// TwinCAT 3 PLC project P1_CompPP
// ProgramVersion: 3.1.4023.0
// libraries:
//   Tc2_Standard, * (Beckhoff Automation GmbH)
//   Tc2_System, * (Beckhoff Automation GmbH)
//   Tc2_Utilities, * (Beckhoff Automation GmbH)
//   Tc3_EventLogger, * (Beckhoff Automation GmbH)
//   Tc3_Module, * (Beckhoff Automation GmbH)
//   Tc2_Utilities,3.3.52.0,Beckhoff Automation GmbH
// project tree:
//   DUTs/ E_ChargerType.TcDUT (not stored), E_State.TcDUT, ST_Alarm_Base.TcDUT (not stored), ST_Charger_Base.TcDUT, ST_ChargeTime.TcDUT (not stored), ST_CSV_Record.TcDUT (not stored), ST_Module.TcDUT, ST_PB_Base.TcDUT (not stored), ST_PrefireDiscon_Base.TcDUT, ST_Segment_Base.TcDUT, ST_Setpoints_Base.TcDUT
//   GVLs/ Alarms_DB.TcGVL (not stored), ChargeTime_DB.TcGVL, csv_DB.TcGVL, EngVal.TcGVL, GVL.TcGVL, HMI_DB.TcGVL, Input.TcGVL, LCP1_IO.TcGVL, LCP2_IO.TcGVL, MCP_IO.TcGVL, Output.TcGVL, Permissives_DB.TcGVL, Setpoints.TcGVL, Trips_DB.TcGVL, VoltMonitor_DB.TcGVL
//   / PlcTask.TcTTO
//   POUs/ ADC_10V.TcPOU, ADC_5V.TcPOU (not stored), Alarms.TcPOU, Alarms_FB.TcPOU (not stored), Alias.TcPOU, AnalogConversion_obs.TcPOU, AnalogConversion.TcPOU, AQ.TcPOU (not stored), ChargeTime.TcPOU, CounterUP.TcPOU, Heartbeat.TcPOU, HMI.TcPOU, LCA_CAL.TcPOU (not stored), MAIN.TcPOU, Norm_x.TcPOU (not stored), Permissives.TcPOU, PermissivesS.TcPOU, plc_plc_comm.TcPOU, RW_CSV.TcPOU (not stored), Sequence_2M.TcPOU, Sequence.TcPOU, Trips.TcPOU, VoltMonitor.TcPOU
//   POUs/csv/ P_ArgToConvExample.TcPOU (not stored), P_StringToConvExample.TcPOU (not stored), P_TextModeRead.TcPOU, P_TextModeWrite_og.TcPOU, P_TextModeWrite.TcPOU
// real-time tasks:
//   TASK PlcTask: cycle T#10ms, priority 20, ADS port 350
// I/O:
//   DEVICE Device 1 (EtherCAT) (disabled), AmsNetId 5.104.171.248.2.1
//     Term 8 (EK1200) [EK1200-5000 EtherCAT Power supply (2A E-Bus)]
//       Term 3 (EL1008) [EL1008 8Ch. Dig. Input 24V, 3ms]
//       Term 4 (EL1008) [EL1008 8Ch. Dig. Input 24V, 3ms]
//       Term 5 (EL1008) [EL1008 8Ch. Dig. Input 24V, 3ms]
//       Term 6 (EL1008) [EL1008 8Ch. Dig. Input 24V, 3ms]
//       Term 14 (EL1008) [EL1008 8Ch. Dig. Input 24V, 3ms]
//       Term 15 (EL2008) [EL2008 8Ch. Dig. Output 24V, 0.5A]
//       Term 16 (EL2008) [EL2008 8Ch. Dig. Output 24V, 0.5A]
//       Term 17 (EL3068) [EL3068 8Ch. Ana. Input 0-10V]
//       Term 18 (EL4008) [EL4008 8Ch. Ana. Output 0-10V, 12bit]
//       Term 18 (EL9011) [EL9011 End Terminal]
//   DEVICE Device 5 (EtherCAT) (disabled), AmsNetId 5.104.171.248.6.1
//     Box 1 (170357) [170357]
//   DEVICE Device 4 (USB) (disabled)
//     Box 2 (C9900-L100 License-Key-USB-Stick)
// variable links:
//   P1_CompPP/P1_CompPP Instance <-> Device 1 (EtherCAT)/Term 8 (EK1200)/Term 14 (EL1008)
//     PlcTask Inputs/Input.R1_05_00 <-> Channel 1/Input
//     PlcTask Inputs/Input.R1_05_01 <-> Channel 2/Input
//     PlcTask Inputs/Input.R1_05_02 <-> Channel 3/Input
//     PlcTask Inputs/Input.R1_05_03 <-> Channel 4/Input
//     PlcTask Inputs/Input.R1_05_04 <-> Channel 5/Input
//     PlcTask Inputs/Input.R1_05_05 <-> Channel 6/Input
//     PlcTask Inputs/Input.R1_05_06 <-> Channel 7/Input
//     PlcTask Inputs/Input.R1_05_07 <-> Channel 8/Input
//   P1_CompPP/P1_CompPP Instance <-> Device 1 (EtherCAT)/Term 8 (EK1200)/Term 15 (EL2008)
//     PlcTask Outputs/Output.R1_06_00 <-> Channel 1/Output
//     PlcTask Outputs/Output.R1_06_01 <-> Channel 2/Output
//     PlcTask Outputs/Output.R1_06_02 <-> Channel 3/Output
//     PlcTask Outputs/Output.R1_06_03 <-> Channel 4/Output
//     PlcTask Outputs/Output.R1_06_04 <-> Channel 5/Output
//     PlcTask Outputs/Output.R1_06_05 <-> Channel 6/Output
//     PlcTask Outputs/Output.R1_06_06 <-> Channel 7/Output
//     PlcTask Outputs/Output.R1_06_07 <-> Channel 8/Output
//   P1_CompPP/P1_CompPP Instance <-> Device 1 (EtherCAT)/Term 8 (EK1200)/Term 16 (EL2008)
//     PlcTask Outputs/Output.R1_07_00 <-> Channel 1/Output
//     PlcTask Outputs/Output.R1_07_01 <-> Channel 2/Output
//     PlcTask Outputs/Output.R1_07_02 <-> Channel 3/Output
//     PlcTask Outputs/Output.R1_07_03 <-> Channel 4/Output
//     PlcTask Outputs/Output.R1_07_04 <-> Channel 5/Output
//     PlcTask Outputs/Output.R1_07_05 <-> Channel 6/Output
//     PlcTask Outputs/Output.R1_07_06 <-> Channel 7/Output
//     PlcTask Outputs/Output.R1_07_07 <-> Channel 8/Output
//   P1_CompPP/P1_CompPP Instance <-> Device 1 (EtherCAT)/Term 8 (EK1200)/Term 17 (EL3068)
//     PlcTask Inputs/Input.R1_08_00 <-> AI Standard Channel 1/Value
//     PlcTask Inputs/Input.R1_08_01 <-> AI Standard Channel 2/Value
//     PlcTask Inputs/Input.R1_08_02 <-> AI Standard Channel 3/Value
//     PlcTask Inputs/Input.R1_08_03 <-> AI Standard Channel 4/Value
//     PlcTask Inputs/Input.R1_08_05 <-> AI Standard Channel 6/Value
//     PlcTask Inputs/Input.R1_08_06 <-> AI Standard Channel 7/Value
//     PlcTask Inputs/Input.R1_08_07 <-> AI Standard Channel 8/Value
//     PlcTask Inputs/Input.R2_08_04 <-> AI Standard Channel 5/Value
//   P1_CompPP/P1_CompPP Instance <-> Device 1 (EtherCAT)/Term 8 (EK1200)/Term 18 (EL4008)
//     PlcTask Outputs/Output.R1_09_00 <-> AO Outputs Channel 1/Analog output
//     PlcTask Outputs/Output.R1_09_01 <-> AO Outputs Channel 2/Analog output
//     PlcTask Outputs/Output.R1_09_02 <-> AO Outputs Channel 3/Analog output
//     PlcTask Outputs/Output.R1_09_03 <-> AO Outputs Channel 4/Analog output
//     PlcTask Outputs/Output.R1_09_04 <-> AO Outputs Channel 5/Analog output
//     PlcTask Outputs/Output.R1_09_05 <-> AO Outputs Channel 6/Analog output
//     PlcTask Outputs/Output.R1_09_06 <-> AO Outputs Channel 7/Analog output
//     PlcTask Outputs/Output.R1_09_07 <-> AO Outputs Channel 8/Analog output
//   P1_CompPP/P1_CompPP Instance <-> Device 1 (EtherCAT)/Term 8 (EK1200)/Term 3 (EL1008)
//     PlcTask Inputs/Input.R1_01_00 <-> Channel 1/Input
//     PlcTask Inputs/Input.R1_01_01 <-> Channel 2/Input
//     PlcTask Inputs/Input.R1_01_02 <-> Channel 3/Input
//     PlcTask Inputs/Input.R1_01_03 <-> Channel 4/Input
//     PlcTask Inputs/Input.R1_01_04 <-> Channel 5/Input
//     PlcTask Inputs/Input.R1_01_05 <-> Channel 6/Input
//     PlcTask Inputs/Input.R1_01_06 <-> Channel 7/Input
//     PlcTask Inputs/Input.R1_01_07 <-> Channel 8/Input
//   P1_CompPP/P1_CompPP Instance <-> Device 1 (EtherCAT)/Term 8 (EK1200)/Term 4 (EL1008)
//     PlcTask Inputs/Input.R1_02_00 <-> Channel 1/Input
//     PlcTask Inputs/Input.R1_02_01 <-> Channel 2/Input
//     PlcTask Inputs/Input.R1_02_02 <-> Channel 3/Input
//     PlcTask Inputs/Input.R1_02_03 <-> Channel 4/Input
//     PlcTask Inputs/Input.R1_02_04 <-> Channel 5/Input
//     PlcTask Inputs/Input.R1_02_05 <-> Channel 6/Input
//     PlcTask Inputs/Input.R1_02_06 <-> Channel 7/Input
//     PlcTask Inputs/Input.R1_02_07 <-> Channel 8/Input
//   P1_CompPP/P1_CompPP Instance <-> Device 1 (EtherCAT)/Term 8 (EK1200)/Term 5 (EL1008)
//     PlcTask Inputs/Input.R1_03_00 <-> Channel 1/Input
//     PlcTask Inputs/Input.R1_03_01 <-> Channel 2/Input
//     PlcTask Inputs/Input.R1_03_02 <-> Channel 3/Input
//     PlcTask Inputs/Input.R1_03_03 <-> Channel 4/Input
//     PlcTask Inputs/Input.R1_03_04 <-> Channel 5/Input
//     PlcTask Inputs/Input.R1_03_05 <-> Channel 6/Input
//     PlcTask Inputs/Input.R1_03_06 <-> Channel 7/Input
//     PlcTask Inputs/Input.R1_03_07 <-> Channel 8/Input
//   P1_CompPP/P1_CompPP Instance <-> Device 1 (EtherCAT)/Term 8 (EK1200)/Term 6 (EL1008)
//     PlcTask Inputs/Input.R1_04_00 <-> Channel 1/Input
//     PlcTask Inputs/Input.R1_04_01 <-> Channel 2/Input
//     PlcTask Inputs/Input.R1_04_02 <-> Channel 3/Input
//     PlcTask Inputs/Input.R1_04_03 <-> Channel 4/Input
//     PlcTask Inputs/Input.R1_04_04 <-> Channel 5/Input
//     PlcTask Inputs/Input.R1_04_05 <-> Channel 6/Input
//     PlcTask Inputs/Input.R1_04_06 <-> Channel 7/Input
//     PlcTask Inputs/Input.R1_04_07 <-> Channel 8/Input
//   P1_CompPP/P1_CompPP Instance <-> Device 5 (EtherCAT)/Box 1 (170357)
//     PlcTask Inputs/Input.B170357_CapRaw[{0..24}] <-> HV Cap process data mapping/Cap {0..24} Raw  (25 links)

CONFIGURATION P1_CompPP
    RESOURCE PLC ON TwinCAT3
        TASK PlcTask(INTERVAL := T#10ms, PRIORITY := 20);
        PROGRAM MAIN WITH PlcTask : MAIN;
        PROGRAM Alias WITH PlcTask : Alias;
    END_RESOURCE
END_CONFIGURATION

// ---- DUTs/E_State.TcDUT
{attribute 'qualified_only'}
{attribute 'strict'}
TYPE E_State :
(
	SAFE			:= 0, //IDLE
	CHARGING		:= 1, //Charge
	CHARGECOMPLETE	:= 2, //EOC
	//DISCONNECTING	:= 3, //Disconnect
	DUMPING			:= 3, 
	ABORT			:= 4,
	TRIPPED			:= 5
);
END_TYPE

// ---- DUTs/ST_Charger_Base.TcDUT
TYPE ST_Charger_Base :
STRUCT
	//DI
	inhibited 		: BOOL;
	EndOfCharge 	: BOOL;
	HV_isON			: BOOL;
	OverTemp		: BOOL;
	InterlockOpen	: BOOL;
	LoadFaulted		: BOOL;
	SummaryFaulted	: BOOL;
	
	//DQ
	inhibit			: BOOL;
	HV_ON			: BOOL;
	
	//AI
	voltageFeedback_raw 	: INT;
	voltageFeedback_norm 	: REAL;
	voltageFeedback			: REAL;
	
	currentFeedback_raw 	: INT;
	currentFeedback_norm	: REAL;
	currentFeedback			: REAL;
	peakCurrent				: REAL;
	
	//AQ
	voltageSP_norm	: REAL;
	voltageSP		: REAL;
	voltageSP_raw	: INT; // setpoint output to field device.
	
	//Internal
	//ChargerType_50kV : BOOL;
	//ChargerType_30kV : BOOL;
	//ChargerType_12kV : BOOL;
	ChargerType		 : INT;
	LossInhibit		 : BOOL;
	LossHVON		 : BOOL;
	LossInhibitTON	 : TON;
	LossHVON_TON	 : TON;
	
	ChargeTime		: ST_ChargeTime;
	
END_STRUCT
END_TYPE

// ---- DUTs/ST_Module.TcDUT
TYPE ST_Module :
STRUCT
	CloseChargeRly	: BOOL;
	OpenDumpRly		: BOOL;
	Fire			: BOOL;
	TriggerScope	: BOOL;
	
	ChargeRly_close	: BOOL;
	DumpRly_open	: BOOL;
	ModuleCharged	: BOOL;
	VoltageFeedback : REAL;
END_STRUCT
END_TYPE

// ---- DUTs/ST_PrefireDiscon_Base.TcDUT
TYPE ST_PrefireDiscon_Base :
STRUCT
	PrefireDisconClosed			: BOOL := FALSE;
	PrefireDisconOpen			: BOOL := FALSE;
	ChargePrefireDisconCap		: BOOL := FALSE;   //1 = charge, 0 = dump?
	ClosePrefireDiscon			: BOOL := FALSE;
END_STRUCT
END_TYPE

// ---- DUTs/ST_Segment_Base.TcDUT
TYPE ST_Segment_Base :
STRUCT
	Module : ARRAY [1..9] OF ST_Module;	
END_STRUCT
END_TYPE

// ---- DUTs/ST_Setpoints_Base.TcDUT
TYPE ST_Setpoints_Base :
STRUCT
	RequiredChargedV : REAL := 12;
	TotalCapacitance : REAL := 10; //uF - LOCAL ONLY, NOT FROM MAIN PLC - LoadCapacitance
	PSratedV		 : REAL := 50;
	wLCA			 : BOOL := TRUE;
	NumOfCharger	 : INT := 1;
	eChargerType		: E_ChargerType;
END_STRUCT
END_TYPE

// ---- GVLs/ChargeTime_DB.TcGVL
{attribute 'qualified_only'}
VAR_GLOBAL RETAIN
	ChargerDelay_TON : ARRAY[1..6] OF TON;
	ChargerDelay_PT  : ARRAY[1..6] OF TIME;
	ChargerDelay_ET  : ARRAY[1..6] OF TIME;	
	
	//SustChargeTime_TON : ARRAY[1..3] OF TON;
	//SustChargeTime_PT  : ARRAY[1..3] OF TIME;
	//SustChargeTime_ET  : ARRAY[1..3] OF TIME;	
	
	//FormChargeTime_TON : ARRAY[1..2] OF TON;
	//FormChargeTime_PT  : ARRAY[1..2] OF TIME;
	//FormChargeTime_ET  : ARRAY[1..2] OF TIME;
	
	LongestChargeTime_TON : TON;
	LongestChargeTime_PT : TIME;
	LongestChargeTime_ET : TIME;

	ChargeTimeStartDelay	: ARRAY[1..6] OF INT; // no SR yet, it will be 7 if SR is added
	ChargingTimeElapse		: ARRAY[1..6] OF INT;	
	ChargingTimeElapse_TON	: ARRAY[1..6] OF TON;
	
	pfcChargerDelay_TON : TON;
	pfcChargerDelay_PT : TIME;
	pfcChargerDelay_ET : TIME;
	
	pfcChargeTimeStartDelay : INT;
	pfcChargingTimeElapse : INT;
	pfcChargingTimeElapse_TON : TON;
END_VAR

// ---- GVLs/csv_DB.TcGVL
{attribute 'qualified_only'}
VAR_GLOBAL
	intDataToCSVINT		: INT;
	realDataToCSVREAL	: REAL;
END_VAR

// ---- GVLs/EngVal.TcGVL
{attribute 'qualified_only'}
VAR_GLOBAL
	Max_50kVChargerVoltage : REAL := 50000; //50kV
	Min_50kVChargerVoltage : REAL := 0;
	
	Max_50kVChargerCurrent : REAL := 0.18; //total peak charge current is 0.18A
	Min_50kVChargerCurrent : REAL := 0;
	
	Max_12kVChargerVoltage : REAL := 12000; //12kV
	Min_12kVChargerVoltage : REAL := 0;
	
	Max_12kVChargerCurrent : REAL := 0.75; //total peak charge current is 0.75A
	Min_12kVChargerCurrent : REAL := 0;
	
	Max_30kVChargerVoltage : REAL := 30000; //30kV
	Min_30kVChargerVoltage : REAL := 0;
	
	Max_30kVChargerCurrent : REAL := 0.6; //total peak charge current is 0.6A
	Min_30kVChargerCurrent : REAL := 0;	
	//Max_GLS1_ChargerV	   : REAL := 50000; //form trigger
	//Max_GLS2_ChargerV	   : REAL := 50000; // preform trigger
	//Max_GLS3_ChargerV	   : REAL := 30000; // preform cap charger
	
	Max_CapVoltage			: REAL := 32000;  //assuming 32kV cap....  
	Min_CapVoltage			: REAL := 0;
	
	UpperLimit12kVCaps		: REAL := 10500; //peak and sust
	//LowerLimit12kVCaps	: REAL := -2000;
	UpperLimit50kVCaps		: REAL := 35000; 
	
	(*ULimit_PeakCapRequiredV	: REAL := 10000; //10kV veto
	LLimit_PeakCapRequiredV	: REAL := -2000; //-2kV
	ULimit_SustCapRequiredV	: REAL := 12000; //12kv veto
	LLimit_SustCapRequiredV	: REAL := -2000; //-2kv
	ULimit_FormCapRequiredV : REAL := 35000;
	LLimit_FormCapRequiredV : REAL := 0;
	*)
	//ULimit_PreFormCapRequiredV : REAL := 30000; //gls3
	//LLimit_PreFormCapRequiredV : REAL := 0;
		
END_VAR

// ---- GVLs/GVL.TcGVL
{attribute 'qualified_only'}
VAR_GLOBAL
	alarm_test	: BOOL;
	test		: BOOL;
	RemoteModeSelected : BOOL;
	
	// %MB ; 4020, %MX; 4021
	WriteStatetoPLC		AT %MB0	: E_State; // write to the pfc plc / 1 = p1 comp pp charge complete, 2 = p1 comp pp dumping
	ReadStateFromPLC	AT %MB2 : E_State;
	pfcChargeTime		AT %MB4	: REAL;
	Button				AT %MB8 : ST_PB_Base; 
END_VAR

VAR_GLOBAL CONSTANT
	MAX_CSV_ROWS 			: UDINT := 500;
	MAX_CSV_COLUMNS 		: UDINT := 2;
	MAX_CSV_FIELD_LENGTH	: UDINT := 150;
END_VAR

// ---- GVLs/HMI_DB.TcGVL
{attribute 'qualified_only'}
VAR_GLOBAL PERSISTENT
	TDKLoad		: ARRAY [1..6] OF ST_Setpoints_Base; //or RETAIN
	
	ChargerHVOFF_rlyDelayPT		: TIME := T#25MS;
	ChargerHVOFF_rlyDelayPT_INT	: INT := 25;
	
	HVONdelayPT					: TIME := T#250MS;
	HVONdelayPT_INT				: INT := 250;
	
	RunOutTMR_PT				: TIME := T#10S;
	RunOutTMR_PT_INT			: DINT := 10;
	RunOutTMR_elapse			: DINT;
	
	ChargingRunOutTMR_elapse	: INT;
	
	FireDelayTMR_TON			: TON;
	FireDelayTMR_PT				: TIME := T#2S;
	FireDelayTMR_ET				: TIME;
	FireDelayTMR_REAL			: REAL := 2;
		
END_VAR

VAR_GLOBAL
	ArmTheCagePB				: BOOL := 0;
	UnArmTheCagePB				: BOOL := 0;
	ChargePB					: BOOL := 0;
	DumpPB						: BOOL := 0;
	AbortPB						: BOOL := 0;
	FirePB						: BOOL := 0;
	ClearFaultPB				: BOOL := 0;
	AllDumpRelaysOpenBP			: BOOL := 0;
	AllChargeRelayCloseBP		: BOOL := 0;
	SystemSafeBP				: BOOL := 0;
	ForceToChargCompletePB		: BOOL := 0;
	
	HMI_ManualModeSelected		: BOOL := 0;  // 1 = manual mode selected
	CloseChargeRlySW			: BOOL := 0;
	OpenDumpRlySW				: BOOL := 0;
	TurnChrgHVonSW				: BOOL := 0;
	TurnChrgInhibitOffSW		: BOOL := 0;
	TurnOnShotTrigSW			: BOOL := 0;
	TurnOnChargeAlarm			: BOOL := 0;
	
	LastTimeShotLog				: BOOL := 0;
	CSV_loggingBusy				: BOOL := 0;
	CSV_loggingError			: BOOL := 0;
	CSV_loggingDone				: BOOL := 0;
	FillingBuffer				: BOOL := 0;
	
	//disconnect
	
	ChargePrefireDisconCap		: BOOL := FALSE;  //1 = charge, 0 = dump?
	ClosePrefireDisconSW		: BOOL := FALSE;
END_VAR

// ---- GVLs/Input.TcGVL
{attribute 'qualified_only'}
VAR_GLOBAL
//***MCP************************************************************************
	//EL1008 - DI1
	R1_01_00 AT	%I*: BOOL; //Master stop PB not pressed - black pb on mcp
	R1_01_01 AT	%I*: BOOL; //case Estop circuit okay (Rly1 (120vac)
	R1_01_02 AT %I*: BOOL; //Remote Mode Selected (NO)
	R1_01_03 AT %I*: BOOL; //MCP PSU1 DC OK
	R1_01_04 AT %I*: BOOL; //Machine Ground Relay Open (lifted) Opto Board
	R1_01_05 AT %I*: BOOL; //spare
	R1_01_06 AT %I*: BOOL; //spare
	R1_01_07 AT %I*: BOOL; //spare

	//EL1008 - DI2
	//TDK802 1
	R1_02_00 AT	%I*: BOOL; //
	R1_02_01 AT	%I*: BOOL;
	R1_02_02 AT %I*: BOOL; 
	R1_02_03 AT %I*: BOOL; 
	R1_02_04 AT %I*: BOOL; 
	R1_02_05 AT %I*: BOOL; 
	R1_02_06 AT %I*: BOOL; 
	R1_02_07 AT %I*: BOOL; //spare
	
	R1_03_00 AT	%I*: BOOL; //
	R1_03_01 AT	%I*: BOOL;
	R1_03_02 AT %I*: BOOL; 
	R1_03_03 AT %I*: BOOL; 
	R1_03_04 AT %I*: BOOL; 
	R1_03_05 AT %I*: BOOL; 
	R1_03_06 AT %I*: BOOL; 
	R1_03_07 AT %I*: BOOL; //spare

	R1_04_00 AT	%I*: BOOL; //
	R1_04_01 AT	%I*: BOOL;
	R1_04_02 AT %I*: BOOL; 
	R1_04_03 AT %I*: BOOL; 
	R1_04_04 AT %I*: BOOL; 
	R1_04_05 AT %I*: BOOL; 
	R1_04_06 AT %I*: BOOL; 
	R1_04_07 AT %I*: BOOL; //spare
	
	R1_05_00 AT	%I*: BOOL; //
	R1_05_01 AT	%I*: BOOL;
	R1_05_02 AT %I*: BOOL; 
	R1_05_03 AT %I*: BOOL; 
	R1_05_04 AT %I*: BOOL; 
	R1_05_05 AT %I*: BOOL; 
	R1_05_06 AT %I*: BOOL; 
	R1_05_07 AT %I*: BOOL; //spare
		
	//EL3068 - AI1
	R1_08_00 		AT %I*: INT;
	R1_08_00_Status AT %I*: WORD;
	
	R1_08_01 		AT %I*: INT;
	R1_08_01_Status AT %I*: WORD;

	R1_08_02 		AT %I*: INT;
	R1_08_02_Status AT %I*: WORD;

	R1_08_03 		AT %I*: INT;
	R1_08_03_Status AT %I*: WORD;

	R2_08_04 		AT %I*: INT;
	R2_08_04_Status AT %I*: WORD;

	R1_08_05 		AT %I*: INT;
	R1_08_05_Status AT %I*: WORD;

	R1_08_06 		AT %I*: INT;
	R1_08_06_Status AT %I*: WORD;

	R1_08_07 		AT %I*: INT;
	R1_08_07_Status AT %I*: WORD;

	//Ethercat Device Voltage
	B170357_CapRaw AT %I* : ARRAY[0..24] OF UINT;
	B170357_BatLevel AT %I* : BOOL;
	B170357_Heartbeat AT %I* : BOOL;
END_VAR

// ---- GVLs/LCP1_IO.TcGVL
{attribute 'qualified_only'}
VAR_GLOBAL
	Segment	: ARRAY [1..3] OF ST_Segment_Base;
END_VAR

// ---- GVLs/LCP2_IO.TcGVL
{attribute 'qualified_only'}
VAR_GLOBAL
	Segment	: ARRAY [4..6] OF ST_Segment_Base;
END_VAR

// ---- GVLs/MCP_IO.TcGVL
{attribute 'qualified_only'}
VAR_GLOBAL
	EStopPB_NotPressed			: BOOL := FALSE;
	DoorSWclose					: BOOL := FALSE;
	EnergizeACKontactor			: BOOL := FALSE;
	ShortContactClose			: BOOL := FALSE;
	UnshortContactClose			: BOOL := FALSE;
	//disconnect
	PrefireDiscon				: ST_PrefireDiscon_Base;
	
	
	//RemoteModeSelected			: BOOL;
	//PSU1_DCOK					: BOOL;
	//MachineGNDrlyOpen			: BOOL;
	//CloseAllChargeRlyCommand	: BOOL; only for slim
	//OpenAllDumpRelayCommand		: BOOL; only for slim
	//Charger 					: ARRAY [1..8] OF ST_Charger_Base;
	//GLS3_Load					: ST_ChargeTime;
	//GLS1_hvON					: BOOL;
	//GLS2_hvON					: BOOL;
	//GLS3_hvON					: BOOL;
	//LiftMachineGND				: BOOL;
	//AllChargeRelaysClose		: BOOL; only for slim
	//AllDumpRelaysOpen			: BOOL; only for slim
	//GLS1_voltageSP				: DINT;
	//GLS1_voltageSP_norm			: REAL;
	//GLS1_voltageSP_raw			: INT;
	
	//GLS2_voltageSP				: DINT;
	//GLS2_voltageSP_norm			: REAL;
	//GLS2_voltageSP_raw			: INT;
	
	//GLS3_voltageSP				: DINT;
	//GLS3_voltageSP_norm			: REAL;
	//GLS3_voltageSP_raw			: INT;

END_VAR

VAR_GLOBAL PERSISTENT
	Charger 					: ARRAY [1..6] OF ST_Charger_Base;
END_VAR

// ---- GVLs/Output.TcGVL
{attribute 'qualified_only'}
VAR_GLOBAL
	//***MCP 
	//EL2008 - DQ1
	R1_06_00 AT %Q*: BOOL;
	R1_06_01 AT %Q*: BOOL;
	R1_06_02 AT %Q*: BOOL;
	R1_06_03 AT %Q*: BOOL;
	R1_06_04 AT %Q*: BOOL;
	R1_06_05 AT %Q*: BOOL;
	R1_06_06 AT %Q*: BOOL;
	R1_06_07 AT %Q*: BOOL;

	//EL2008 - DQ1
	R1_07_00 AT %Q*: BOOL;
	R1_07_01 AT %Q*: BOOL;
	R1_07_02 AT %Q*: BOOL;
	R1_07_03 AT %Q*: BOOL;
	R1_07_04 AT %Q*: BOOL;
	R1_07_05 AT %Q*: BOOL;
	R1_07_06 AT %Q*: BOOL;
	R1_07_07 AT %Q*: BOOL;
	
	//EL4008 - AQ1
	R1_09_00 AT %Q*: INT;	//Charger 1 - Voltage Setpoint
	R1_09_01 AT %Q*: INT;	//Charger 2 - Voltage Setpoint
	R1_09_02 AT %Q*: INT;	//Charger 3 - Voltage Setpoint
	R1_09_03 AT %Q*: INT;	//Charger 4 - Voltage Setpoint
	R1_09_04 AT %Q*: INT;	//Charger 5 - Voltage Setpoint	
	R1_09_05 AT %Q*: INT;	//Charger 6 - Voltage Setpoint	
	R1_09_06 AT %Q*: INT;	//spare
	R1_09_07 AT %Q*: INT;	//spare
	
END_VAR

// ---- GVLs/Permissives_DB.TcGVL
{attribute 'qualified_only'}
VAR_GLOBAL
	CageInterlockOK			: BOOL := 0;
	ShortingSystemEngaged	: BOOL := 0;
	AllChargerEOC			: BOOL := 0;
	AllChargeRelayClosed	: BOOL := 0;
	AllDumpRelayOpen		: BOOL := 0;
	ReadyToCharge			: BOOL := 0;
	PrefireDisconClosed		: BOOL := FALSE;
	PreFireDisconOpen		: BOOL := FALSE;
END_VAR

// ---- GVLs/Setpoints.TcGVL
{attribute 'qualified_only'}
VAR_GLOBAL
	TDKLoad : ARRAY [1..6] OF ST_Setpoints_Base;
	
	
END_VAR

// ---- GVLs/Trips_DB.TcGVL
{attribute 'qualified_only'}
VAR_GLOBAL
		
	//AnyEstopPressed 			: BOOL;
	//AllDCpsuOK					: BOOL;
	//AnyChargerOverTemp			: BOOL;
	//AnyChargerLoadFault			: BOOL;
	//AnyChargerInterlockOpen		: BOOL;
	//AnyChargerFaulted			: BOOL; // same as summary fault
	
	//SystemTripped 				: BOOL;
	//InstrumentationFaulted		: BOOL;
	//AnyChargeRlyFail			: BOOL;
	//AnyDumpRlyFail				: BOOL;
	//AnyACInterlockFail			: BOOL;
	//AnyLossInhibitSignal		: BOOL;
	//AnyLossHVONsignal			: BOOL;
	
	ChargingTimerRunout         : BOOL;
	ChargedTimerRunout			: BOOL;
	DumpTimerRunout				: BOOL;
	//SystemTimeOut				: BOOL;
	NoFaultDetected				: BOOL;
	TimerRunOutON				: BOOL;
	
	ChargerSummaryFault			: BOOL;
	
	EStopPBpressed				: BOOL;
	CageDoorNotClose			: BOOL;
	ShortingSystemUnknown		: BOOL;
	PrefireDisconUnknown		: BOOL;
END_VAR

// ---- GVLs/VoltMonitor_DB.TcGVL
{attribute 'qualified_only'}
VAR_GLOBAL
	Heartbeat : BOOL;
	BateryOn  : BOOL;
	BatteryLow : BOOL := 0;
	Channel	: USINT; //ST_AnalogCHSelection;
	VoltageReading_raw : ARRAY[0..24] OF INT; //custom board
	VoltageReading_norm : ARRAY[0..24] OF REAL;
	VoltageReading	: ARRAY[0..15] OF REAL;
	LoadMaxRatedV	: REAL := 13800; //-2k TO 35kV
	LoadMinRatedV	: REAL := -1450; //Jake's lab result
//***************************************
	CapRaw : ARRAY[0..24] OF UINT;
	CapRawBIT : STRING;
	CapRaw_DummySnap : ARRAY[0..24] OF UINT;
	CapRaw_Str: STRING;
	BatteryLevel : BOOL;
	
	//cunter for missing packets
	missedCTU : CTU;
	//ONS	: R_TRIG;
	missingCNT : WORD :=0;
	LossVoltMonitorBoard : BOOL := 0;
//**********************************	
	Time1		: TON;
	Time1_ET	: TIME;
	packetsPerMin : REAL;
	//missedCTU : CTU;
	ONS	: R_TRIG;
	//missingCNT : WORD;
	missingCNT_REAL : REAL;
END_VAR

// ---- POUs/MAIN.TcPOU
PROGRAM MAIN
VAR
END_VAR

Alias();
plc_plc_comm(); //comment this out if not talking to pfc
Permissives();
Trips();
ChargeTime();
AnalogConversion();
VoltMonitor();
Sequence();
HMI();
Heartbeat();
Alarms();
RW_CSV(); // to use this, you would need to create a folder directory in the PLC C drive

END_PROGRAM

// ---- POUs/Alias.TcPOU
PROGRAM Alias
VAR
	i : INT := 0;
END_VAR

 //R1 : MCP**  
	
//INPUT
	//DI	
	MCP_IO.EStopPB_NotPressed					:= Input.R1_01_00;  //NC - 
	MCP_IO.DoorSWclose							:= Input.R1_01_01;  
	MCP_IO.ShortContactClose					:= Input.R1_01_02; 
	MCP_IO.UnshortContactClose					:= Input.R1_01_03; 
	//MCP_IO.MachineGNDrlyOpen					:= Input.R1_01_04; // machine ground lifted (opto board)	
	//MCP_IO.CloseAllChargeRlyCommand				:= Input.R1_01_05; // command from screen room (opto) - Slim only
	//MCP_IO.OpenAllDumpRelayCommand				:= Input.R1_01_06; // command from screen room (opto) - slim only

	//DI
	MCP_IO.Charger[1].inhibited					:= NOT Input.R1_02_00; //TDK802 1 NC for all feedback esaigeean
	MCP_IO.Charger[1].EndOfCharge				:= NOT Input.R1_02_01; //TDK802 1
	MCP_IO.Charger[1].HV_isON					:= NOT Input.R1_02_02; //TDK802 1
	MCP_IO.Charger[1].SummaryFaulted			:= NOT Input.R1_02_03; //TDK802 1
	//MCP_IO.Charger[1].OverTemp					:= Input.R1_02_03; //TDK802 1
	//MCP_IO.Charger[1].InterlockOpen				:= Input.R1_02_04; //TDK802 1
	//MCP_IO.Charger[1].LoadFaulted				:= Input.R1_02_05; //TDK802 1

	LCP1_IO.Segment[1].Module[1].ChargeRly_close := Input.R1_02_04;
	LCP1_IO.Segment[1].Module[1].DumpRly_open	 := NOT Input.R1_02_05;
	
	//prefire disconn	
	MCP_IO.PrefireDiscon.PrefireDisconClosed	:= Input.R1_03_00;
	MCP_IO.PrefireDiscon.PrefireDisconOpen		:= Input.R1_03_01;
	
	//EL3068 - AI
	MCP_IO.Charger[1].voltageFeedback_raw		:= Input.R1_08_00;
	MCP_IO.Charger[1].currentFeedback_raw		:= Input.R1_08_01;
	
	//OUTPUT
	//DQ
	Output.R1_06_00	:= MCP_IO.Charger[1].inhibit;
	Output.R1_06_01	:= MCP_IO.Charger[1].HV_ON;
	Output.R1_06_02	:= LCP1_IO.Segment[1].Module[1].CloseChargeRly;
	Output.R1_06_03	:= LCP1_IO.Segment[1].Module[1].OpenDumpRly;
	Output.R1_06_04	:= LCP1_IO.Segment[1].Module[1].Fire;
	Output.R1_06_05	:= LCP1_IO.Segment[1].Module[1].TriggerScope;
	Output.R1_06_06	:= MCP_IO.EnergizeACKontactor;
	Output.R1_06_07	:= LCP1_IO.Segment[1].Module[1].ModuleCharged;
	
	Output.R1_07_00	:= MCP_IO.PrefireDiscon.ChargePrefireDisconCap;
	Output.R1_07_01	:= MCP_IO.PrefireDiscon.ClosePrefireDiscon;							
	
	
	//AQ
	Output.R1_09_00								:= MCP_IO.Charger[1].voltageSP_raw;
	
	//Cap voltage monitor feedback is at VoltMonitor
	VoltMonitor_DB.CapRaw[0] 					:= Input.B170357_CapRaw[0]; 
	
	FOR i := 1 TO 24 BY 1 DO 
		VoltMonitor_DB.CapRaw[i] 					:= Input.B170357_CapRaw[i]; 
	END_FOR
	
IF i > 24 THEN
	i := 1; // make it to 0
END_IF
	
//*************************************************************************************************************

END_PROGRAM

// ---- POUs/plc_plc_comm.TcPOU
PROGRAM plc_plc_comm
VAR
//	WritetoPLC	: ADSwrite_FB;
	ReadStatusfromPLC		: ADSREAD;
	ReadChargTimefromPLC	: ADSREAD;
//	ReadVariableTMR_TON : TON;
	WritetoPLC				: ADSWRITE;
	WriteFireButtontoPLC	: ADSWRITE;
	WriteVariableTMR_TON 	: TON;
	ReadVariableTMR_TON 	: TON;
END_VAR

// also add this to the plc 18Moudle program
//ReadVariableTMR_TON(IN := NOT ReadVariableTMR_TON.Q, PT := T#10MS);
ReadVariableTMR_TON(IN := NOT ReadVariableTMR_TON.Q, PT := T#10MS);
WriteVariableTMR_TON(IN := NOT WriteVariableTMR_TON.Q, PT := T#10MS);

//WritetoPLC (NETID   := '192.168.173.70', //'5.107.220.56.1.1',- pfc plc
WritetoPLC (NETID   := '5.107.220.56.1.1', //- pfc plc
    		PORT    := 851,
    		IDXGRP  := 16#4020,
    		IDXOFFS := 16#0000,
    		LEN     := SIZEOF(GVL.WriteStatetoPLC), //*MB0
    		SRCADDR := ADR(GVL.WriteStatetoPLC),
    		WRITE   := WriteVariableTMR_TON.Q,
    		TMOUT   := T#1S,
			);
			
WriteFireButtontoPLC (NETID   := '5.107.220.56.1.1', //- pfc plc
    		PORT    := 851,
    		IDXGRP  := 16#4020,
    		IDXOFFS := 16#0008,
    		LEN     := SIZEOF(GVL.Button.FirePBPressed), //*MB0
    		SRCADDR := ADR(GVL.Button.FirePBPressed),
    		WRITE   := WriteVariableTMR_TON.Q,
    		TMOUT   := T#1S,
			);	
		
ReadStatusfromPLC (NETID 	:= '5.107.220.56.1.1', //p1 pp plc addr 
			PORT 	:= 851,
			IDXGRP 	:= 16#4020,
			IDXOFFS	:= 16#2, 
			LEN		:= SIZEOF(GVL.ReadStateFromPLC), //*MB2
			DESTADDR:= ADR(GVL.ReadStateFromPLC),
			READ	:= ReadVariableTMR_TON.Q, //high - starts reading
			TMOUT	:= T#2S,
			);
			
ReadChargTimefromPLC (NETID 	:= '5.107.220.56.1.1', //p1 pp plc addr 
			PORT 	:= 851,
			IDXGRP 	:= 16#4020,
			IDXOFFS	:= 16#4, 
			LEN		:= SIZEOF(GVL.pfcChargeTime), //*MB2
			DESTADDR:= ADR(GVL.pfcChargeTime),
			READ	:= ReadVariableTMR_TON.Q, //high - starts reading
			TMOUT	:= T#2S,
			);

END_PROGRAM

// ---- POUs/Permissives.TcPOU
PROGRAM Permissives
VAR
	//AllChargeRelayClosed 	: BOOL := 0;
	//AllDumpRelayOpen		: BOOL := 0;
	//ReadyToCharge			: BOOL := 0;
	//AllChargerEOC			: BOOL := 0;
	
	ChargerVBelowThres		: BOOL := 0;
	ChargedVThres			: REAL := 50;
	AllChargerHVisOFF		: BOOL := 0;
	AllChargerInhibitON		: BOOL := 0;

	AllCapsDischarged		: BOOL := 0;
	SystemIsSafe			: BOOL := 0;
	
END_VAR

IF MCP_IO.ShortContactClose = TRUE AND MCP_IO.UnshortContactClose = FALSE THEN 
	Permissives_DB.ShortingSystemEngaged := TRUE;
	ELSIF MCP_IO.ShortContactClose = FALSE AND MCP_IO.UnshortContactClose = TRUE THEN
		Permissives_DB.ShortingSystemEngaged := FALSE;
END_IF


IF MCP_IO.DoorSWclose = TRUE AND MCP_IO.EStopPB_NotPressed = TRUE THEN 
	Permissives_DB.CageInterlockOK := TRUE;
	ELSE
		Permissives_DB.CageInterlockOK := FALSE;
	END_IF

IF Permissives_DB.CageInterlockOK = FALSE OR HMI_DB.UnArmTheCagePB = TRUE THEN 
	MCP_IO.EnergizeACKontactor := FALSE;
END_IF

IF LCP1_IO.Segment[1].Module[1].ChargeRly_close = TRUE(*AND all the other modules *) OR HMI_DB.AllChargeRelayCloseBP = TRUE
	THEN
		Permissives_DB.AllChargeRelayClosed := TRUE;
	ELSE
		Permissives_DB.AllChargeRelayClosed := FALSE;
END_IF;

IF LCP1_IO.Segment[1].Module[1].DumpRly_open = TRUE(*AND all the other modules *) OR HMI_DB.AllDumpRelaysOpenBP = TRUE
	THEN
		Permissives_DB.AllDumpRelayOpen := TRUE;
	ELSIF LCP1_IO.Segment[1].Module[1].DumpRly_open = FALSE THEN
		Permissives_DB.AllDumpRelayOpen := FALSE;
END_IF;

IF Permissives_DB.AllChargeRelayClosed = TRUE AND Permissives_DB.AllDumpRelayOpen = TRUE THEN
	Permissives_DB.ReadyToCharge := TRUE;
	ELSE 
		Permissives_DB.ReadyToCharge := FALSE;
END_IF

IF MCP_IO.Charger[1].voltageFeedback <= 20 (*AND all other Chargers*) THEN
	ChargerVBelowThres := TRUE;
	ELSE
		ChargerVBelowThres := FALSE;
END_IF;

IF MCP_IO.Charger[1].HV_isON = FALSE (*AND all other Chargers*) THEN
	AllChargerHVisOFF := TRUE;
	ELSE 
		AllChargerHVisOFF := FALSE;
END_IF

IF MCP_IO.Charger[1].inhibited = TRUE (*AND all other Chargers*) THEN
	AllChargerInhibitON	:= TRUE;
	ELSE
		AllChargerInhibitON	:= FALSE;
END_IF;

//Cap voltage feedback
IF (LCP1_IO.Segment[1].Module[1].VoltageFeedback <= ChargedVThres) AND 
	(LCP1_IO.Segment[1].Module[1].VoltageFeedback >= -ChargedVThres) AND 
	(VoltMonitor_DB.CapRaw[0] <> 0)(*  AND all other module voltage feedback <= 50 *) THEN
	AllCapsDischarged := TRUE;
	LCP1_IO.Segment[1].Module[1].ModuleCharged := FALSE; //for status light only
	ELSE 
		AllCapsDischarged := FALSE;
END_IF


IF (ChargerVBelowThres = TRUE AND 
	//AllChargerHVisOFF = TRUE AND 
	//AllChargerInhibitON	= TRUE AND 
	Permissives_DB.AllDumpRelayOpen = FALSE AND 
	AllCapsDischarged = TRUE AND 
	Permissives_DB.CageInterlockOK = TRUE) OR HMI_DB.SystemSafeBP = TRUE
THEN
	(*MCP_IO.Charger[2].voltageFeedback <= 10 AND *)
	SystemIsSafe := TRUE;
	ELSE
		SystemIsSafe := FALSE;
END_IF


IF MCP_IO.Charger[1].EndOfCharge = TRUE (*AND
	MCP_IO.Charger[2].EndOfCharge = TRUE AND
	MCP_IO.Charger[3].EndOfCharge = TRUE AND
	MCP_IO.Charger[4].EndOfCharge = TRUE AND
	MCP_IO.Charger[5].EndOfCharge = TRUE AND
	MCP_IO.Charger[6].EndOfCharge = TRUE *)
THEN
	Permissives_DB.AllChargerEOC := TRUE;
	ELSE
		Permissives_DB.AllChargerEOC := FALSE;

END_IF;

//prefire disconn
IF MCP_IO.PrefireDiscon.PrefireDisconClosed = TRUE AND MCP_IO.PrefireDiscon.PrefireDisconOpen = FALSE THEN 
	Permissives_DB.PrefireDisconClosed := TRUE;
	ELSE
		Permissives_DB.PrefireDisconClosed := FALSE;
END_IF

IF MCP_IO.PrefireDiscon.PrefireDisconClosed = FALSE AND MCP_IO.PrefireDiscon.PrefireDisconOpen = TRUE THEN 
	Permissives_DB.PrefireDisconOpen := TRUE;
	ELSE
		Permissives_DB.PrefireDisconOpen := FALSE;
END_IF

IF (MCP_IO.PrefireDiscon.PrefireDisconClosed = TRUE AND MCP_IO.PrefireDiscon.PrefireDisconOpen = TRUE) OR 
	(MCP_IO.PrefireDiscon.PrefireDisconClosed = FALSE AND MCP_IO.PrefireDiscon.PrefireDisconOpen = FALSE) 
	THEN 
		Trips_DB.PrefireDisconUnknown := TRUE;
		ELSE
			Trips_DB.PrefireDisconUnknown := FALSE;
END_IF

END_PROGRAM

// ---- POUs/Trips.TcPOU
PROGRAM Trips
VAR
	ContactDelay_TON : TON;
	ContactDelay_PT	: TIME:= T#2S;
	ContactDelay_ET	: TIME;
END_VAR

Trips_DB.CageDoorNotClose 		:= NOT MCP_IO.DoorSWclose;
Trips_DB.ChargerSummaryFault 	:= MCP_IO.Charger[1].SummaryFaulted;
Trips_DB.EStopPBpressed 		:= NOT MCP_IO.EStopPB_NotPressed;

IF (MCP_IO.ShortContactClose = TRUE AND MCP_IO.UnshortContactClose = TRUE) OR 
	(MCP_IO.ShortContactClose = FALSE AND MCP_IO.UnshortContactClose = FALSE)
	THEN
		ContactDelay_TON(IN := TRUE, PT := ContactDelay_PT, ET => ContactDelay_ET);
		ELSE
			ContactDelay_TON(IN := FALSE);
END_IF

IF ContactDelay_TON.Q = TRUE THEN 
	Trips_DB.ShortingSystemUnknown := TRUE;
	ContactDelay_TON(IN := FALSE);
END_IF

END_PROGRAM

// ---- POUs/ChargeTime.TcPOU
PROGRAM ChargeTime
VAR

	lca_charge_cal	 : ARRAY [1..6] OF LCA_CAL;
	i				 : INT := 1; // 1-8 instances
	j				 : INT := 1; //1 - 8 ch
	m				 : INT := 1;
	n				 : INT := 6; // no SR here yet
	a				 : INT := 1; 
	
	Q				 : REAL := 1; // Charge
	Current			 : REAL := 0.1; //100mA
	
	longestChargeTime: REAL;
	
END_VAR

//mapping hmi input to setpoints
FOR j := 1 TO n BY 1 DO	
	Setpoints.TDKLoad[j].TotalCapacitance	:= HMI_DB.TDKLoad[j].TotalCapacitance;
	Setpoints.TDKLoad[j].PSratedV 			:= HMI_DB.TDKLoad[j].PSratedV;
	Setpoints.TDKLoad[j].RequiredChargedV	:= HMI_DB.TDKLoad[j].RequiredChargedV;  
	Setpoints.TDKLoad[j].wLCA				:= HMI_DB.TDKLoad[j].wLCA;
	Setpoints.TDKLoad[j].NumOfCharger		:= HMI_DB.TDKLoad[j].NumOfCharger;	
	
	//charge time delay and elapse for HMI
	ChargeTime_DB.ChargeTimeStartDelay[j] := TIME_TO_INT((ChargeTime_DB.ChargerDelay_PT[j] - ChargeTime_DB.ChargerDelay_ET[j])/1000);
	ChargeTime_DB.ChargingTimeElapse[j] := TIME_TO_INT((ChargeTime_DB.ChargingTimeElapse_TON[j].PT - ChargeTime_DB.ChargingTimeElapse_TON[j].ET)/1000);
END_FOR

//ChargeTime_DB.PreFormChargeTimeStartDelay := TIME_TO_INT((ChargeTime_DB.PreFormChargeTime_PT - ChargeTime_DB.PreFormChargeTime_ET)/1000);
//ChargeTime_DB.PreFormChargingTimeElapse := TIME_TO_INT((ChargeTime_DB.PreFormChargingTimeElapse_TON.PT - ChargeTime_DB.PreFormChargingTimeElapse_TON.ET)/1000);

(*
//GLS 3
Setpoints.GLSLoad.TotalCapacitance	:= HMI_DB.GLSLoad.TotalCapacitance;
Setpoints.GLSLoad.PSratedV 			:= HMI_DB.GLSLoad.PSratedV;
//Setpoints.PreFormBank.RequiredChargedV	:= Recipe.PreFormBank.RequiredChargedV; //only thing that comes from the main plc recipe
//Setpoints.GLSLoad.wLCA				:= HMI_DB.GLSLoad.wLCA;
Setpoints.GLSLoad.NumOfCharger		:= HMI_DB.GLSLoad.NumOfCharger;	
*)


//veto
//this should not happen
FOR m := 1 TO n BY 1 DO
	IF Setpoints.TDKLoad[m].RequiredChargedV <= -2 THEN
		Setpoints.TDKLoad[m].RequiredChargedV := -2;
	END_IF	
END_FOR

(*
//charger 1 is 30kV*********************************************
IF 1000*(Setpoints.TDKLoad[1].RequiredChargedV) >= 12000 THEN
			Setpoints.TDKLoad[1].RequiredChargedV := (10000/1000); //limit at 10kv
			HMI_DB.TDKLoad[1].RequiredChargedV := (10000/1000);
	ELSIF Setpoints.TDKLoad[1].RequiredChargedV <= 0 THEN
			Setpoints.TDKLoad[1].RequiredChargedV := 0;
			HMI_DB.TDKLoad[1].RequiredChargedV := 0;
END_IF
//charger 1 is 30kV*********************************************
*)
//from 2 to 6
FOR i := 1 TO n BY 1 DO
	IF MCP_IO.Charger[i].ChargerType = E_ChargerType.TDK50kV THEN 
		//set limites of charger voltage input from HMI input
		IF 1000*(Setpoints.TDKLoad[i].RequiredChargedV) >= EngVal.UpperLimit50kVCaps THEN
			Setpoints.TDKLoad[i].RequiredChargedV := (EngVal.UpperLimit50kVCaps/1000); //limit at 35kv
			HMI_DB.TDKLoad[i].RequiredChargedV := (EngVal.UpperLimit50kVCaps/1000);
		ELSIF Setpoints.TDKLoad[i].RequiredChargedV <= 0 THEN
			Setpoints.TDKLoad[i].RequiredChargedV := 0;
			HMI_DB.TDKLoad[i].RequiredChargedV := 0;
		END_IF
	ELSIF MCP_IO.Charger[i].ChargerType = E_ChargerType.TDK12kV OR MCP_IO.Charger[i].ChargerType = E_ChargerType.TDK30kV THEN
		//set limites of charger voltage input from HMI input
		IF 1000*(Setpoints.TDKLoad[i].RequiredChargedV) >= EngVal.UpperLimit12kVCaps THEN
			Setpoints.TDKLoad[i].RequiredChargedV := (EngVal.UpperLimit12kVCaps/1000); //limit at 10kv
			HMI_DB.TDKLoad[i].RequiredChargedV := (EngVal.UpperLimit12kVCaps/1000); //limit at 10kv
		ELSIF Setpoints.TDKLoad[i].RequiredChargedV <= 0 THEN
			Setpoints.TDKLoad[i].RequiredChargedV := ABS(Setpoints.TDKLoad[i].RequiredChargedV);
			HMI_DB.TDKLoad[i].RequiredChargedV := ABS(Setpoints.TDKLoad[i].RequiredChargedV);
		END_IF
	END_IF;
END_FOR;
(*//ch 1 - 3
IF Setpoints.TDKLoad[1].RequiredChargedV >= 10 THEN
	Setpoints.TDKLoad[1].RequiredChargedV := 10;
	ELSIF Setpoints.TDKLoad[1].RequiredChargedV < 0 THEN
		Setpoints.TDKLoad[1].RequiredChargedV := ABS(Setpoints.TDKLoad[1].RequiredChargedV); 
END_IF
IF Setpoints.TDKLoad[2].RequiredChargedV >= 10 THEN
	Setpoints.TDKLoad[2].RequiredChargedV := 10;
	ELSIF Setpoints.TDKLoad[2].RequiredChargedV < 0 THEN
		Setpoints.TDKLoad[2].RequiredChargedV := ABS(Setpoints.TDKLoad[2].RequiredChargedV); 	
END_IF
IF Setpoints.TDKLoad[3].RequiredChargedV >= 10 THEN
	Setpoints.TDKLoad[3].RequiredChargedV := 10;
	ELSIF Setpoints.TDKLoad[3].RequiredChargedV < 0 THEN
		Setpoints.TDKLoad[3].RequiredChargedV := ABS(Setpoints.TDKLoad[3].RequiredChargedV); 	
END_IF

//ch 4-6
IF Setpoints.TDKLoad[4].RequiredChargedV >= 12 THEN
	Setpoints.TDKLoad[4].RequiredChargedV := 12;
	ELSIF Setpoints.TDKLoad[4].RequiredChargedV < 0 THEN
		Setpoints.TDKLoad[4].RequiredChargedV := ABS(Setpoints.TDKLoad[4].RequiredChargedV); 	
END_IF
IF Setpoints.TDKLoad[5].RequiredChargedV >= 12 THEN
	Setpoints.TDKLoad[5].RequiredChargedV := 12;
	ELSIF Setpoints.TDKLoad[5].RequiredChargedV < 0 THEN
		Setpoints.TDKLoad[5].RequiredChargedV := ABS(Setpoints.TDKLoad[5].RequiredChargedV); 	
END_IF
IF Setpoints.TDKLoad[6].RequiredChargedV >= 12 THEN
	Setpoints.TDKLoad[6].RequiredChargedV := 12;
	ELSIF Setpoints.TDKLoad[6].RequiredChargedV < 0 THEN
		Setpoints.TDKLoad[6].RequiredChargedV := ABS(Setpoints.TDKLoad[6].RequiredChargedV); 	
END_IF
*)

//chg time
FOR i := 1 TO n BY 1 DO
	lca_charge_cal[i](	PSratedV := Setpoints.TDKLoad[i].PSratedV, 
						RequiredChargeV := Setpoints.TDKLoad[i].RequiredChargedV, 
						LoadCapacitance := Setpoints.TDKLoad[i].TotalCapacitance, 
						NumOfCharger := Setpoints.TDKLoad[i].NumOfCharger, 
						wLCA := Setpoints.TDKLoad[i].wLCA
						);

	MCP_IO.Charger[i].ChargeTime.timeToChargeLoad := lca_charge_cal[i].TimeToChargeLoad;
	MCP_IO.Charger[i].ChargeTime.Power := lca_charge_cal[i].RespectedPower;
	
	IF Setpoints.TDKLoad[i].RequiredChargedV = 0 THEN
		MCP_IO.Charger[i].ChargeTime.timeToChargeLoad := 0;
		MCP_IO.Charger[i].ChargeTime.Power := 0;
	END_IF
END_FOR



(*
//gls - gls3 is preform cap charger
Q := 1000* Setpoints.GLSLoad.RequiredChargedV * (Setpoints.GLSLoad.TotalCapacitance / 1000000);
MCP_IO.GLS3_Load.timeToChargeLoad := Q / Current;
MCP_IO.GLS3_Load.Power := 1000*Setpoints.GLSLoad.RequiredChargedV * Current;
*)
//find the longest charge time.  //need more work
longestChargeTime := MAX( MCP_IO.Charger[1].ChargeTime.timeToChargeLoad,
							MCP_IO.Charger[2].ChargeTime.timeToChargeLoad,
							MCP_IO.Charger[3].ChargeTime.timeToChargeLoad,
							MCP_IO.Charger[4].ChargeTime.timeToChargeLoad,
							MCP_IO.Charger[5].ChargeTime.timeToChargeLoad,
							MCP_IO.Charger[6].ChargeTime.timeToChargeLoad,
							//MCP_IO.Charger[7].ChargeTime.timeToChargeLoad, //no SR yet
							GVL.pfcChargeTime
							(*MCP_IO.Charger[7].ChargeTime.timeToChargeLoad,
							MCP_IO.Charger[8].ChargeTime.timeToChargeLoad, *)
							(*MCP_IO.GLS3_Load.timeToChargeLoad*));

ChargeTime_DB.LongestChargeTime_PT := REAL_TO_TIME (1000*longestChargeTime);

//FOR a := 1 TO 8 BY 1 DO
FOR a := 1 TO n BY 1 DO
	IF (longestChargeTime - MCP_IO.Charger[a].ChargeTime.timeToChargeLoad) >= 0 THEN
		ChargeTime_DB.ChargerDelay_PT[a] := REAL_TO_TIME (1000*(longestChargeTime - MCP_IO.Charger[a].ChargeTime.timeToChargeLoad));
		ELSE 
			ChargeTime_DB.ChargerDelay_PT[a] := REAL_TO_TIME (1000*(MCP_IO.Charger[a].ChargeTime.timeToChargeLoad - longestChargeTime));
	END_IF;		

	//IF (longestChargeTime - MCP_IO.Charger[a+3].ChargeTime.timeToChargeLoad) >= 0 THEN
	//	ChargeTime_DB.SustChargeTime_PT[a] := REAL_TO_TIME (1000*(longestChargeTime - MCP_IO.Charger[a+3].ChargeTime.timeToChargeLoad));	
	//END_IF;	
	
END_FOR;

		
IF (longestChargeTime - GVL.pfcChargeTime)>= 0 THEN 
	ChargeTime_DB.pfcChargerDelay_PT := REAL_TO_TIME (1000*(longestChargeTime - GVL.pfcChargeTime));
	ELSE
		ChargeTime_DB.pfcChargerDelay_PT := REAL_TO_TIME (1000*(GVL.pfcChargeTime - longestChargeTime));	
END_IF

(*IF (longestChargeTime - MCP_IO.Charger[7].ChargeTime.timeToChargeLoad) >= 0 THEN
	ChargeTime_DB.FormChargeTime_PT[1] := REAL_TO_TIME (1000*(longestChargeTime - MCP_IO.Charger[7].ChargeTime.timeToChargeLoad));	
END_IF;	
IF (longestChargeTime - MCP_IO.Charger[8].ChargeTime.timeToChargeLoad) >= 0 THEN
	ChargeTime_DB.FormChargeTime_PT[2] := REAL_TO_TIME (1000*(longestChargeTime - MCP_IO.Charger[8].ChargeTime.timeToChargeLoad));	
END_IF;	

IF (longestChargeTime - MCP_IO.GLS3_Load.timeToChargeLoad) >= 0 THEN
		ChargeTime_DB.PreFormChargeTime_PT := REAL_TO_TIME (1000*(longestChargeTime - MCP_IO.GLS3_Load.timeToChargeLoad));
		ELSE
			ChargeTime_DB.PreFormChargeTime_PT := REAL_TO_TIME (1000*(MCP_IO.GLS3_Load.timeToChargeLoad -longestChargeTime));
END_IF;
*)


//IF i > 8 THEN 
IF i > n THEN 
	i := 1;
END_IF

IF j > n THEN
	j := 1;
END_IF

IF m > n THEN
	m := 1;
END_IF

//IF a > 8 THEN
IF a > n THEN
	a := 1;
END_IF;

END_PROGRAM

// ---- POUs/AnalogConversion.TcPOU
PROGRAM AnalogConversion
VAR
	i					: INT := 1; //charger 1-6
	j					: INT := 1;  // section 1 - 4 
	k					: INT := 1;  // cap 1-10
	m					: INT := 1; //form cap 1-12
	eChargerType 		: E_ChargerType;
	
END_VAR

//MCP Charger 
//Analog Input
FOR i := 1 TO 6 BY 1 DO 
	//MCP_IO.Charger[i].voltageSP := (HMI_DB.TDKLoad[i].RequiredChargedV *1000);
	MCP_IO.Charger[i].voltageSP := (1000*Setpoints.TDKLoad[i].RequiredChargedV);
END_FOR
(*
//charger 1 is 30kV *************************************************************************************
																					
//*************************************************************************************
*)


//AI
FOR i := 1 TO 6 BY 1 DO
	//voltage
	MCP_IO.Charger[i].voltageFeedback_norm := Norm_x (raw_input := INT_TO_REAL (MCP_IO.Charger[i].voltageFeedback_raw),
														x_max := 32767,
														x_min := 0);
	//current																									
	MCP_IO.Charger[i].currentFeedback_norm := Norm_x (raw_input := INT_TO_REAL (MCP_IO.Charger[i].currentFeedback_raw),
														x_max := 32767,
														x_min := 0);
							
	//50kV chargers feedback
	//if 50kV config selected
	IF MCP_IO.Charger[i].ChargerType = E_ChargerType.TDK50kV THEN 
		//50kv
		MCP_IO.Charger[i].voltageFeedback := (EngVal.Max_50kVChargerVoltage - EngVal.Min_50kVChargerVoltage) * ADC_10V(
																							normal_input := MCP_IO.Charger[i].voltageFeedback_norm,
																							x_max := 10,
																							x_min := 0);
		//peak current scaling
		IF Setpoints.TDKLoad[i].wLCA = TRUE THEN 
			MCP_IO.Charger[i].peakCurrent := EngVal.Max_50kVChargerCurrent*2;
			ELSE 
				MCP_IO.Charger[i].peakCurrent := EngVal.Max_50kVChargerCurrent;
		END_IF	
		MCP_IO.Charger[i].currentFeedback := (MCP_IO.Charger[i].peakCurrent - EngVal.Min_50kVChargerCurrent) * ADC_10V(
																							normal_input := MCP_IO.Charger[i].currentFeedback_norm,
																							x_max := 10,
																							x_min := 0);
		//12kv
	ELSIF MCP_IO.Charger[i].ChargerType = E_ChargerType.TDK12kV THEN
		MCP_IO.Charger[i].voltageFeedback := (EngVal.Max_12kVChargerVoltage - EngVal.Min_12kVChargerVoltage) * ADC_10V(
																							normal_input := MCP_IO.Charger[i].voltageFeedback_norm,
																							x_max := 10,
																							x_min := 0);
		//peak current scaling
		IF Setpoints.TDKLoad[i].wLCA = TRUE THEN 
			MCP_IO.Charger[i].peakCurrent := 2.17; //EngVal.Max_12kVChargerCurrent*2; //1.5A - this para is uncalibrated, from experiment, it is 2.17
			ELSE 
				MCP_IO.Charger[i].peakCurrent := 2.17; //EngVal.Max_12kVChargerCurrent;
		END_IF
		MCP_IO.Charger[i].currentFeedback := (MCP_IO.Charger[i].peakCurrent - EngVal.Min_12kVChargerCurrent) * ADC_10V(
																							normal_input := MCP_IO.Charger[i].currentFeedback_norm,
																							x_max := 10,
																							x_min := 0);	
	ELSIF MCP_IO.Charger[i].ChargerType = E_ChargerType.TDK30kV THEN
		MCP_IO.Charger[i].voltageFeedback := (EngVal.Max_30kVChargerVoltage - EngVal.Min_30kVChargerVoltage) * ADC_10V(
																							normal_input := MCP_IO.Charger[i].voltageFeedback_norm,
																							x_max := 10,
																							x_min := 0);														
		//peak current scaling
		IF Setpoints.TDKLoad[i].wLCA = TRUE THEN 
			MCP_IO.Charger[i].peakCurrent := EngVal.Max_30kVChargerCurrent*2;// 1.2A
			ELSE 
				MCP_IO.Charger[i].peakCurrent := EngVal.Max_30kVChargerCurrent;
		END_IF
		// 30kV charger max current output is 0.6A													
		MCP_IO.Charger[i].currentFeedback := (MCP_IO.Charger[i].peakCurrent - EngVal.Min_30kVChargerCurrent) * ADC_10V(
																							normal_input := MCP_IO.Charger[i].currentFeedback_norm,
																							x_max := 10,
																							x_min := 0);							
	END_IF;	
END_FOR;

//Analog Output
//voltageSP = Required Charge Voltage**

(*
//prepare output signal for 30kV chargers.  //**Setpoints.RequiredChargedV -> MCP_IO.Charger.voltageSP **
MCP_IO.Charger[1].voltageSP_norm := Norm_x (raw_input := (MCP_IO.Charger[1].voltageSP), 
												x_max := (HMI_DB.TDKLoad[1].PSratedV * 1000),
												x_min := 0);
		
MCP_IO.Charger[1].voltageSP_raw := AQ (norm_input := MCP_IO.Charger[1].voltageSP_norm, 
												x_max := 10,
												x_min := 0); 


//prepare output signal for 30kV chargers.  //**Setpoints.RequiredChargedV -> MCP_IO.Charger.voltageSP **
MCP_IO.Charger[1].voltageSP_norm := Norm_x (raw_input := (MCP_IO.Charger[1].voltageSP), 
												x_max := HMI_DB.TDKLoad[1].PSratedV,
												x_min := 0);
		
MCP_IO.Charger[1].voltageSP_raw := AQ (norm_input := MCP_IO.Charger[1].voltageSP_norm, 
												x_max := 10,
												x_min := 0); 

//Charger 1 is 30kV *************************************
IF MCP_IO.Charger[1].voltageSP >= (12000) THEN
			MCP_IO.Charger[1].voltageSP := 10000; //limit at 35kV
		ELSIF MCP_IO.Charger[1].voltageSP <= 0 THEN
			MCP_IO.Charger[1].voltageSP := 0; //limit at 0V
		END_IF; 

												
//limite for output sigal (<= 10V)  this should not happen
//IF MCP_IO.Charger[1].voltageSP_raw >= 32767 THEN 
//	MCP_IO.Charger[1].voltageSP_raw := 32767; 										
//END_IF;
//*******************************************************
*)	
//FOR i := 1 TO 8 BY 1 DO
FOR i := 1 TO 6 BY 1 DO	
	
	//if 50kV config selected
	IF MCP_IO.Charger[i].ChargerType = E_ChargerType.TDK50kV THEN 
		//set limits of charger voltage input 
		IF MCP_IO.Charger[i].voltageSP >= (EngVal.UpperLimit50kVCaps) THEN
			MCP_IO.Charger[i].voltageSP := 35000; //limit at 35kV
		ELSIF MCP_IO.Charger[i].voltageSP <= 0 THEN
			MCP_IO.Charger[i].voltageSP := 0; //limit at 0V
		END_IF; 
		
		//prepare output signal for 50kV chargers.
		MCP_IO.Charger[i].voltageSP_norm := Norm_x (raw_input :=(MCP_IO.Charger[i].voltageSP), 
												x_max := EngVal.Max_50kVChargerVoltage,
												x_min := EngVal.Min_50kVChargerVoltage);	
												
		MCP_IO.Charger[i].voltageSP_raw := AQ (norm_input := MCP_IO.Charger[i].voltageSP_norm, 
												x_max := 10,
												x_min := 0);
												
	ELSIF MCP_IO.Charger[i].ChargerType = E_ChargerType.TDK12kV THEN 
		//set limits of charger voltage input 
		IF MCP_IO.Charger[i].voltageSP >= (EngVal.UpperLimit12kVCaps) THEN
			MCP_IO.Charger[i].voltageSP := 10500; //limit at 35kV
		ELSIF MCP_IO.Charger[i].voltageSP <= 0 THEN
			MCP_IO.Charger[i].voltageSP := ABS(MCP_IO.Charger[i].voltageSP); //limit at 0V
		END_IF; 
		
		//prepare output signal for 50kV chargers.
		MCP_IO.Charger[i].voltageSP_norm := Norm_x (raw_input :=(MCP_IO.Charger[i].voltageSP), 
												x_max := EngVal.Max_12kVChargerVoltage,
												x_min := EngVal.Min_12kVChargerVoltage);	
												
		MCP_IO.Charger[i].voltageSP_raw := AQ (norm_input := MCP_IO.Charger[i].voltageSP_norm, 
												x_max := 10,
												x_min := 0);
	
	ELSIF MCP_IO.Charger[i].ChargerType = E_ChargerType.TDK30kV THEN 		
		//set limits of charger voltage input 
		IF MCP_IO.Charger[i].voltageSP >= (EngVal.UpperLimit12kVCaps) THEN
			MCP_IO.Charger[i].voltageSP := 10500; //limit at 35kV
		ELSIF MCP_IO.Charger[i].voltageSP <= 0 THEN
			MCP_IO.Charger[i].voltageSP := ABS(MCP_IO.Charger[i].voltageSP); //limit at 0V
		END_IF;
		//prepare output signal for 30kV chargers.
		MCP_IO.Charger[i].voltageSP_norm := Norm_x (raw_input :=(MCP_IO.Charger[i].voltageSP), 
												x_max := EngVal.Max_30kVChargerVoltage,
												x_min := EngVal.Min_30kVChargerVoltage);	
												
		MCP_IO.Charger[i].voltageSP_raw := AQ (norm_input := MCP_IO.Charger[i].voltageSP_norm, 
												x_max := 10,
												x_min := 0);
	END_IF;	
												
	//limite for output sigal (<= 10V)  this should not happen
	IF MCP_IO.Charger[i].voltageSP_raw >= 32767 THEN 
		MCP_IO.Charger[i].voltageSP_raw := 32767; 										
	END_IF;
	
END_FOR;

//Cap voltage feedback
//IF Input.B170357_CapRaw[0] <> 0 THEN
															//can also add a range of x samples for self calibrating
	VoltMonitor_DB.VoltageReading_norm[0] := Norm_x (raw_input := INT_TO_REAL (VoltMonitor_DB.VoltageReading_raw[0]),
														x_max := 904, //10bit value - 1110001000 = 904deci
														x_min := 100); //100deci is the zero of range -1.61 to 12.01
	LCP1_IO.Segment[1].Module[1].VoltageFeedback := (12010 - 0) * ADC_10V(normal_input := VoltMonitor_DB.VoltageReading_norm[0],
																		x_max := 12.01,
																		x_min := 0); //use zero, it will cal for the -ve	

IF VoltMonitor.DataNull = TRUE THEN
	LCP1_IO.Segment[1].Module[1].VoltageFeedback := NULL;
END_IF


//reset counter
//IF i > 8 THEN
IF i > 6 THEN
	i := 1;
END_IF;

IF j > 3 THEN 
	j := 1;
END_IF

IF k > 10 THEN 
	k := 1;
END_IF

IF m > 12 THEN 
	m := 1;
END_IF

END_PROGRAM

// ---- POUs/ADC_10V.TcPOU
FUNCTION ADC_10V : REAL
VAR_INPUT
	normal_input : REAL;
	x_max : REAL := 10;
	x_min : REAL := 0;
END_VAR
VAR
	voltage_reading : REAL;
END_VAR

// 0 - 10V AI INPUT | normal_input 0-100%
voltage_reading := x_max * normal_input;
ADC_10V := (voltage_reading - x_min) / (x_max - x_min);

//voltage_reading := normal_input * (x_max - x_min);
//ADC_10V := voltage_reading / (x_max - x_min);

END_FUNCTION

// ---- POUs/VoltMonitor.TcPOU
PROGRAM VoltMonitor
VAR
	i : USINT := 0;
	k : USINT := 0;
	counter : USINT := 0;
	b : ARRAY[0..3] OF BOOL;
	b1 : BOOL;
	b2 : BOOL;
	b3 : BOOL;
	pause : BOOL;
	VMBoardWDT_TON : TON;
	VMBoardWDT_PT	: TIME := T#2S;
	VMBoardWDT_ET	: TIME;
	DataNull	: BOOL := 0;
	DataNullRebunceTMR_TON : TON;
	DataNullRebounce_PT	: TIME := T#800MS;
END_VAR


(*IF Heartbeat.pulse_ms = TRUE AND pause = FALSE THEN
	i := i + 1;
	counter := 16-i;
	IF counter >= 16 THEN 
		counter := 0;
	END_IF
	VoltMonitor_DB.Channel := counter ;
	VoltMonitor_DB.VoltageReading_raw[counter] := GVL.raw_VoltageMonitor;
END_IF*)

b[0] := 0; //VoltMonitor_DB.Channel.0;
b[1] := 0; //VoltMonitor_DB.Channel.1;
b[2] := 0; //VoltMonitor_DB.Channel.2;
b[3] := 0; //VoltMonitor_DB.Channel.3;
//VoltMonitor_DB.VoltageReading_raw[0] := GVL.raw_VoltageMonitor;


//VoltMonitor_DB.CapRaw_Str :=  MID (UINT_TO_STRING (GVL.B170357_CapRaw), 10, 5);



//VoltMonitor_DB.VoltageReading_raw[0] := VoltMonitor_DB.CapRaw; //STRING_TO_INT (VoltMonitor_DB.CapRaw_Str);
FOR k := 0 TO 1 BY 1 DO //0 - 1 two channels only
	
	IF Input.B170357_CapRaw[k] <> 0 THEN
		VoltMonitor_DB.VoltageReading_raw[k].0 := VoltMonitor_DB.CapRaw[k].2;
		VoltMonitor_DB.VoltageReading_raw[k].1 := VoltMonitor_DB.CapRaw[k].3;
		VoltMonitor_DB.VoltageReading_raw[k].2 := VoltMonitor_DB.CapRaw[k].4;
		VoltMonitor_DB.VoltageReading_raw[k].3 := VoltMonitor_DB.CapRaw[k].5;
	
		VoltMonitor_DB.VoltageReading_raw[k].4 := VoltMonitor_DB.CapRaw[k].6;
		VoltMonitor_DB.VoltageReading_raw[k].5 := VoltMonitor_DB.CapRaw[k].7;
		VoltMonitor_DB.VoltageReading_raw[k].6 := VoltMonitor_DB.CapRaw[k].8;
		VoltMonitor_DB.VoltageReading_raw[k].7 := VoltMonitor_DB.CapRaw[k].9;
	
		VoltMonitor_DB.VoltageReading_raw[k].8 := VoltMonitor_DB.CapRaw[k].10;
		VoltMonitor_DB.VoltageReading_raw[k].9 := VoltMonitor_DB.CapRaw[k].11;
	
		VoltMonitor_DB.VoltageReading_raw[k].10 := 0;//VoltMonitor_DB.CapRaw.14;
		VoltMonitor_DB.VoltageReading_raw[k].11 := 0;//VoltMonitor_DB.CapRaw.15;
		VoltMonitor_DB.VoltageReading_raw[k].12 := 0;//VoltMonitor_DB.CapRaw.12;
		VoltMonitor_DB.VoltageReading_raw[k].13 := 0;//VoltMonitor_DB.CapRaw.13;
		VoltMonitor_DB.VoltageReading_raw[k].14 := 0; //VoltMonitor_DB.CapRaw.14;
	
		VoltMonitor_DB.VoltageReading_raw[k].15 := 0;//VoltMonitor_DB.CapRaw.4;
		//VoltMonitor_DB.CapRaw_DummySnap[k] := Input.B170357_CapRaw[k];//VoltMonitor_DB.VoltageReading_raw[0];
		//ELSE
		//	VoltMonitor_DB.VoltageReading_raw[k] := ULINT_TO_INT(NULL);
			//VoltMonitor_DB.CapRaw_DummySnap[k] := 0;
	END_IF
	
END_FOR

VoltMonitor_DB.BatteryLow := VoltMonitor_DB.CapRaw[0].13;

IF VoltMonitor_DB.CapRaw[0] = 0 THEN 
	VMBoardWDT_TON (IN := TRUE, PT := VMBoardWDT_PT, ET => VMBoardWDT_ET);
	ELSE 
		VMBoardWDT_TON (IN := FALSE);
END_IF

IF VMBoardWDT_TON.Q THEN 
	DataNull := TRUE; 
	VoltMonitor_DB.LossVoltMonitorBoard := TRUE;
END_IF

IF DataNull = TRUE THEN
	VoltMonitor_DB.VoltageReading_raw[0] := ULINT_TO_INT(NULL);
END_IF

IF VoltMonitor_DB.LossVoltMonitorBoard = TRUE THEN
	DataNullRebunceTMR_TON( IN := TRUE, PT := DataNullRebounce_PT);
END_IF

IF DataNullRebunceTMR_TON.Q = TRUE THEN
	DataNull := FALSE;
	DataNullRebunceTMR_TON( IN := FALSE);
END_IF



//VoltMonitor_DB.CapRawBIT := WORD_TO_HEXSTR ( UINT_TO_WORD( VoltMonitor_DB.CapRaw[0] ), iPrecision := 16, bLoCase := FALSE);
VoltMonitor_DB.CapRawBIT := BYTE_TO_BINSTR( UINT_TO_BYTE( VoltMonitor_DB.CapRaw[0] ), iPrecision := 16);
//missedCTU.PV := 10000;
//missedCTU.RESET := FALSE;
(*
IF Input.B170357_CapRaw[1] <> Input.B170357_CapRaw[11] OR 
	Input.B170357_CapRaw[2] <> Input.B170357_CapRaw[12] OR 
	Input.B170357_CapRaw[2] <> Input.B170357_CapRaw[13] OR 
	Input.B170357_CapRaw[3] <> Input.B170357_CapRaw[14] OR 
	Input.B170357_CapRaw[3] <> Input.B170357_CapRaw[15] OR 
	Input.B170357_CapRaw[1] <> Input.B170357_CapRaw[16] //OR 
	(*GVL.B170357_CapRaw[1] <> GVL.B170357_CapRaw[13]*) THEN
	VoltMonitor_DB.missedCTU.CU := TRUE;
	//VoltMonitor_DB.ONS (CLK := TRUE);
	ELSE
		VoltMonitor_DB.missedCTU.CU := FALSE;
		//VoltMonitor_DB.ONS.CLK := FALSE; 
END_IF

VoltMonitor_DB.missingCNT_REAL := WORD_TO_REAL(VoltMonitor_DB.missingCNT);
CounterUP();
*)
//missingCNT := missedCTU.CV;

//IF pause = TRUE THEN
//	VoltMonitor_DB.VoltageReading_raw[0] := 0;
//END_IF;

IF i > 16 THEN 
	i := 0;
END_IF

IF k > 1 THEN 
	k := 0;
END_IF

END_PROGRAM

// ---- POUs/CounterUP.TcPOU
PROGRAM CounterUP
VAR

END_VAR

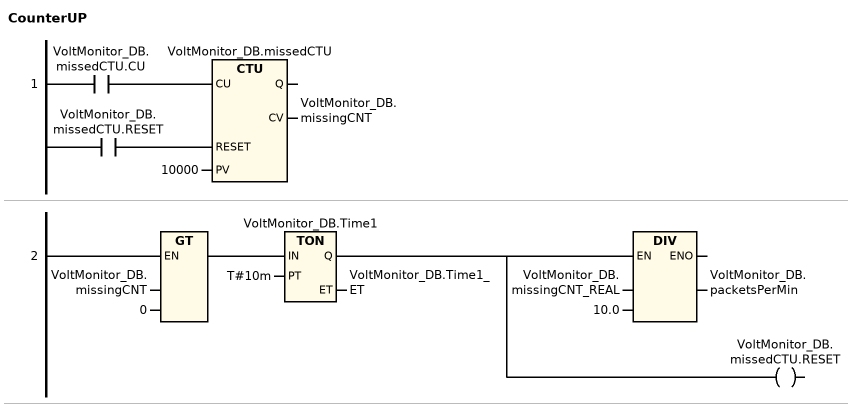
// NETWORK 1
VoltMonitor_DB.missedCTU(
    CU := VoltMonitor_DB.missedCTU.CU,
    RESET := VoltMonitor_DB.missedCTU.RESET,
    PV := 10000,
    CV => VoltMonitor_DB.missingCNT); // CTU

// NETWORK 2
VoltMonitor_DB.Time1(IN := VoltMonitor_DB.missingCNT > 0, PT := T#10m, ET => VoltMonitor_DB.Time1_ET); // TON
IF VoltMonitor_DB.Time1.Q THEN VoltMonitor_DB.packetsPerMin := VoltMonitor_DB.missingCNT_REAL / 10.0; END_IF
VoltMonitor_DB.missedCTU.RESET := VoltMonitor_DB.Time1.Q;

END_PROGRAM

// ---- POUs/Sequence.TcPOU
PROGRAM Sequence  //make sure the change the name to Sequence when we use it for the HMI bitmappings.
VAR
	//This sequence is for with PFC. - change the naming non Sequence when it is not used
	eState : E_State;
	
	ChargeRlyDelayON_Timer  : TON;
	ChargeRlyDelayDONE		: BOOL;
	ChargeRlyDelayON_PT		: TIME := T#250MS; //used for delay close and delay open for safe mode
	AbortPSnRlyDelay_Timer	: TON;
	AbortPSnRlyDelay_PT		: TIME := T#5MS; //defualt is 5ms
	AbortPSnRlyDelayDONE	: BOOL;
	ChargeCompleted			: BOOL;
	ChargingRunOutTMR_TON	: TON;
	ChargingRunOutTMR_ET	: TIME;
	ChargedRunOutTMR_TON	: TON;
	ChargedRunOutTMR_ET		: TIME;
	FireToSafeDelayTMR_TON	: TON;
	FireToSafeDelayTMR_PT	: TIME := T#5S;
	FireToSafeDelayTMR_ET	: TIME;
	FirePBpressed			: BOOL := FALSE;
	ShotFired				: BOOL := FALSE;
	
	ShotTrigDelayTMR_TON	: LTON;
	ShotTrigDelayTMR_PT		: LTIME := LTIME#10US;
	ShotTrigDelayTMR_ET		: LTIME;
	
	ShotTrigPulseTMR_TON	: LTON;
	ShotTrigPulseTMR_PT		: LTIME := LTIME#1S + ShotTrigDelayTMR_PT;
	ShotTrigPulseTMR_ET		: LTIME;
		
	ScopeTrigPulseTMR_TON	: LTON;
	ScopeTrigPulseTMR_PT	: LTIME := LTIME#10US;
	ScopeTrigPulseTMR_ET	: LTIME;
	
	DumpingRunOutTMR_TON 	: TON;
	DumpingRunOutTMR_PT		: TIME := T#20S;
	DumpingRunOutTMR_ET		: TIME;
	LocalDumpActive			: BOOL := FALSE;

	StartChargingBroadcast	: BOOL := FALSE;
	StartCharger			: ARRAY[1..8] OF BOOL;
	n						: INT := 8; // number of chargers skip 7, 8 is the pfc
	ChargeTimeFinished		: BOOL;
	StartCharWarningTMR_TON : TON;
	StartCharWarningTMR_PT	: TIME := T#5S;
	StartCharWarningTMR_ET	: TIME;
	ChargeDelayStart		: BOOL;

	
	i						: INT := 1;
	m						: INT := 1;
END_VAR


//Critical Delay Time
HMI_DB.ChargerHVOFF_rlyDelayPT := INT_TO_TIME(HMI_DB.ChargerHVOFF_rlyDelayPT_INT);
AbortPSnRlyDelay_PT := HMI_DB.ChargerHVOFF_rlyDelayPT;

//hv output delay
HMI_DB.HVONdelayPT := INT_TO_TIME (HMI_DB.HVONdelayPT_INT);
ChargeRlyDelayON_PT := HMI_DB.HVONdelayPT;

//runout timer
HMI_DB.RunOutTMR_PT := DINT_TO_TIME (HMI_DB.RunOutTMR_PT_INT*1000);
HMI_DB.RunOutTMR_elapse := (TIME_TO_DINT (HMI_DB.RunOutTMR_PT - ChargedRunOutTMR_TON.ET))/1000;
HMI_DB.ChargingRunOutTMR_elapse := TIME_TO_INT(ChargingRunOutTMR_TON.PT/1000 - ChargingRunOutTMR_TON.ET/1000);

//charge realy timer 
ChargeRlyDelayON_Timer(PT := ChargeRlyDelayON_PT);

//reset timer
IF eState <> E_State.CHARGING THEN 
	ChargingRunOutTMR_TON (IN := FALSE);
	//LCP1_IO.Segment[1].Module[1].ModuleCharged := FALSE; //for status light only

	FOR i := 1 TO 6 BY 1 DO
		ChargeTime_DB.ChargerDelay_TON[i] (IN := FALSE, PT := ChargeTime_DB.ChargerDelay_PT[i], ET => ChargeTime_DB.ChargerDelay_ET[i]);
		ChargeTime_DB.ChargingTimeElapse_TON[i].IN := FALSE;
		ChargeRlyDelayON_Timer (IN := FALSE);
	END_FOR;
	ChargeTime_DB.pfcChargerDelay_TON (IN := FALSE, PT := ChargeTime_DB.pfcChargerDelay_PT, ET => ChargeTime_DB.pfcChargerDelay_ET);
	
	ChargeTime_DB.pfcChargingTimeElapse_TON.IN := FALSE;
END_IF

IF eState <> E_State.CHARGECOMPLETE THEN 
	//LCP1_IO.Segment[1].Module[1].ModuleCharged := FALSE; //for status light only
	ChargedRunOutTMR_TON (IN := FALSE); // only needed in charge complete
END_IF

IF HMI_DB.HMI_ManualModeSelected = TRUE AND eState = E_State.SAFE THEN
	eState := E_State.ManualMode;
END_IF

IF eState = E_State.CHARGING OR eState = E_State.CHARGECOMPLETE OR eState = E_State.ABORT THEN
	HMI_DB.HMI_ManualModeSelected := FALSE;
END_IF

//if not in manual mode turn off the switches
IF eState <> E_State.ManualMode THEN
	HMI_DB.CloseChargeRlySW := FALSE;
	HMI_DB.OpenDumpRlySW := FALSE;
	HMI_DB.TurnChrgHVonSW := FALSE;
	HMI_DB.TurnChrgInhibitOffSW := FALSE;
	HMI_DB.TurnOnShotTrigSW := FALSE;
	HMI_DB.TurnOnChargeAlarm := FALSE;
	HMI_DB.ClosePrefireDisconSW := FALSE;
	HMI_DB.ChargePrefireDisconCap := FALSE;
END_IF

IF HMI_DB.DumpPB = TRUE THEN
	eState := E_State.DUMPING;
	ELSIF HMI_DB.AbortPB = TRUE OR Trips_DB.TimerRunOutON = TRUE OR Permissives_DB.CageInterlockOK = FALSE THEN 
		eState := E_State.ABORT;
	//	ELSE
	//		eState := E_State.SAFE;
		END_IF;

CASE eState OF 
	
	//Safe OR IDLE
	E_State.SAFE:
		ChargeCompleted := FALSE;
		FirePBpressed := FALSE;
		
		FireToSafeDelayTMR_TON (IN := FALSE);
		
		ChargingRunOutTMR_TON (IN := FALSE);
		ChargedRunOutTMR_TON (IN := FALSE);
		DumpingRunOutTMR_TON (IN := FALSE);
		
		ShotTrigDelayTMR_TON (IN := FALSE, PT := ShotTrigDelayTMR_PT, ET => ShotTrigDelayTMR_ET);
		ScopeTrigPulseTMR_TON (IN := FALSE, PT := ScopeTrigPulseTMR_PT, ET => ScopeTrigPulseTMR_ET);
		ShotTrigPulseTMR_TON (IN := FALSE, PT := ShotTrigPulseTMR_PT, ET => ShotTrigPulseTMR_ET);
		
		ChargeTime_DB.LongestChargeTime_TON (IN := FALSE); //reset timer
		ChargeRlyDelayON_Timer ( IN := FALSE, PT := ChargeRlyDelayON_PT);
		ChargeTimeFinished := FALSE; //reset chargetime done bit
		LCP1_IO.Segment[1].Module[1].Fire := FALSE; //turn off all firing triggers
		
		//prefire disconn
		MCP_IO.PrefireDiscon.ChargePrefireDisconCap := FALSE;
		MCP_IO.PrefireDiscon.ClosePrefireDiscon	:= FALSE; //leave disconn open
		
		GVL.WriteStatetoPLC := E_state.SAFE; //status to pfc PP
		
		IF Permissives_DB.CageInterlockOK = TRUE AND HMI_DB.ArmTheCagePB = TRUE THEN 
			MCP_IO.EnergizeACKontactor := TRUE;
		END_IF;
		//HMI_DB.CloseChargeRlySW := FALSE;
		//HMI_DB.OpenDumpRlySW := FALSE;
		
		//TURN OFF ALL CHARGERS
		FOR i := 1 TO 6 BY 1 DO 
			MCP_IO.Charger[i].inhibit := TRUE; // inhibit = high, no output | inhibit = low, allows output
			MCP_IO.Charger[i].HV_ON := FALSE; 
			//MCP_IO.Charger[i].voltageSP := 0.001;
			StartCharger[i] := FALSE; // reset bit
			ChargeTimeFinished := FALSE;
			StartChargingBroadcast := FALSE;
			//reset charger delay timer
			ChargeTime_DB.ChargerDelay_TON[i] (IN := FALSE, PT := ChargeTime_DB.ChargerDelay_PT[i], ET => ChargeTime_DB.ChargerDelay_ET[i]);
			ChargeTime_DB.ChargingTimeElapse_TON[i] (IN := FALSE); 
		END_FOR;
		//pfc
		StartCharger[8] := FALSE;
		ChargeTime_DB.pfcChargerDelay_TON (IN := FALSE, PT := ChargeTime_DB.pfcChargerDelay_PT, ET => ChargeTime_DB.pfcChargerDelay_ET);

		LCP1_IO.Segment[1].Module[1].CloseChargeRly := FALSE;
		LCP1_IO.Segment[1].Module[2].CloseChargeRly := FALSE;
		LCP1_IO.Segment[1].Module[3].CloseChargeRly := FALSE;
		
		LCP1_IO.Segment[1].Module[1].OpenDumpRly := FALSE;
		LCP1_IO.Segment[1].Module[2].OpenDumpRly := FALSE;
		LCP1_IO.Segment[1].Module[3].OpenDumpRly := FALSE;
		
		//when charge pb is pressed
		IF HMI_DB.ChargePB = TRUE AND MCP_IO.EnergizeACKontactor = TRUE AND Permissives_DB.PreFireDisconOpen = TRUE THEN
			ChargeDelayStart := TRUE;
		ELSIF HMI_DB.DumpPB = TRUE THEN
				eState := E_State.DUMPING; 
		END_IF;
		
		IF ChargeDelayStart = TRUE THEN
			// turn on warning light  - do it for all i and j
			LCP1_IO.Segment[1].Module[1].ModuleCharged := TRUE;
			StartCharWarningTMR_TON (IN := TRUE, PT := StartCharWarningTMR_PT, ET=> StartCharWarningTMR_ET);
		END_IF;
		
		IF StartCharWarningTMR_TON.Q = TRUE THEN 
			ChargeDelayStart := FALSE;
			eState := E_State.CHARGING;
		END_IF

	E_State.CHARGING:
	
		//start charging the disconnect cap
		//MCP_IO.PrefireDiscon.ChargePrefireDisconCap := TRUE; //no more capacitor - using ssv
	
		ChargeDelayStart := FALSE;
		StartCharWarningTMR_TON (IN := FALSE, PT := StartCharWarningTMR_PT, ET=> StartCharWarningTMR_ET);
		// turn on warning light  - do it for all i and j
		LCP1_IO.Segment[1].Module[1].ModuleCharged := TRUE;
		
		FirePBpressed := FALSE;
		LCP1_IO.Segment[1].Module[1].Fire := FALSE; //make sure it is off
		//start charging runout timer
		LCP1_IO.Segment[1].Module[1].CloseChargeRly := TRUE;
		LCP1_IO.Segment[1].Module[2].CloseChargeRly := TRUE;
		LCP1_IO.Segment[1].Module[3].CloseChargeRly := TRUE;
		
		LCP1_IO.Segment[1].Module[1].OpenDumpRly := TRUE;
		LCP1_IO.Segment[1].Module[2].OpenDumpRly := TRUE;
		LCP1_IO.Segment[1].Module[3].OpenDumpRly := TRUE;
		
		GVL.WriteStatetoPLC := E_state.CHARGING; //status to pfc PP
		
		IF Permissives_DB.ReadyToCharge = TRUE THEN 
			FOR i := 1 TO 6 BY 1 DO 
				//MCP_IO.Charger[i].voltageSP := (HMI_DB.TDKLoad[i].RequiredChargedV *1000);
				MCP_IO.Charger[i].voltageSP := (1000*HMI_DB.TDKLoad[i].RequiredChargedV);
			END_FOR
		END_IF;
		//start charging runout timer
		ChargingRunOutTMR_TON (IN := TRUE, PT := (ChargeTime_DB.LongestChargeTime_PT + HMI_DB.RunOutTMR_PT), ET => ChargingRunOutTMR_ET);
		
		IF Trips_DB.ChargingTimerRunout = TRUE THEN 
			StartChargingBroadcast := FALSE; // reset the broadcast bit whne all chargers
			ChargeTimeFinished := FALSE; //reset chargetime done bit
			ChargingRunOutTMR_TON (IN := FALSE);
			FOR i := 1 TO 6 BY 1 DO 
				ChargeTime_DB.ChargingTimeElapse_TON[i] (IN := FALSE);							
			END_FOR
			
			eState := E_State.ABORT; 
		END_IF
		
		IF Permissives_DB.AllChargeRelayClosed = TRUE THEN
			//start broadcasting on charger timer
			StartChargingBroadcast := TRUE;
		END_IF;
		//start timer 
		IF StartChargingBroadcast = TRUE THEN 
			//start total charge time TIMER
			ChargeTime_DB.LongestChargeTime_TON (IN := TRUE, PT := ChargeTime_DB.LongestChargeTime_PT, ET => ChargeTime_DB.LongestChargeTime_ET);
			
			//mapping HMI Charger Voltage SP to MCP IO 
			(*FOR i := 1 TO 6 BY 1 DO
				MCP_IO.Charger[i].voltageSP :=(HMI_DB.TDKLoad[i].RequiredChargedV * 1000);
				//MCP_IO.Charger[1].voltageSP := REAL_TO_DINT (Setpoints.TDKLoad[1].RequiredChargedV);
			END_FOR;*)
			
			// delay stagger starts here
			ChargeTime_DB.ChargerDelay_TON[1] (IN := TRUE, PT := ChargeTime_DB.ChargerDelay_PT[1], ET => ChargeTime_DB.ChargerDelay_ET[1]);
			ChargeTime_DB.ChargerDelay_TON[2] (IN := TRUE, PT := ChargeTime_DB.ChargerDelay_PT[2], ET => ChargeTime_DB.ChargerDelay_ET[2]);
			ChargeTime_DB.ChargerDelay_TON[3] (IN := TRUE, PT := ChargeTime_DB.ChargerDelay_PT[3], ET => ChargeTime_DB.ChargerDelay_ET[3]);
		
			ChargeTime_DB.ChargerDelay_TON[4] (IN := TRUE, PT := ChargeTime_DB.ChargerDelay_PT[4], ET => ChargeTime_DB.ChargerDelay_ET[4]);
			ChargeTime_DB.ChargerDelay_TON[5] (IN := TRUE, PT := ChargeTime_DB.ChargerDelay_PT[5], ET => ChargeTime_DB.ChargerDelay_ET[5]);
			ChargeTime_DB.ChargerDelay_TON[6] (IN := TRUE, PT := ChargeTime_DB.ChargerDelay_PT[6], ET => ChargeTime_DB.ChargerDelay_ET[6]);
			//pfc
			ChargeTime_DB.pfcChargerDelay_TON (IN := TRUE, PT := ChargeTime_DB.pfcChargerDelay_PT, ET => ChargeTime_DB.pfcChargerDelay_ET);
			ELSE
				//Turn inhibit High on all chargers and turn off all timer if no broadcasting
				FOR i := 1 TO 6 BY 1 DO 
					MCP_IO.Charger[i].inhibit := TRUE; 
					MCP_IO.Charger[i].HV_ON := FALSE;
					// turn off timer
					ChargeTime_DB.ChargerDelay_TON[i] (IN := FALSE, PT := ChargeTime_DB.ChargerDelay_PT[i], ET => ChargeTime_DB.ChargerDelay_ET[i]);
				END_FOR;
				//pfc
				ChargeTime_DB.pfcChargerDelay_TON (IN := FALSE, PT := ChargeTime_DB.pfcChargerDelay_PT, ET => ChargeTime_DB.pfcChargerDelay_ET);
		END_IF;
			
		FOR i := 1 TO 6 BY 1 DO	
			//turn on HV output to load	
			IF ChargeTime_DB.ChargerDelay_TON[i].Q = TRUE THEN
				StartCharger[i] := TRUE;
			END_IF	
			
			IF StartCharger[i] = TRUE (*AND Permissives.ReadyToCharge = TRUE*) THEN
				MCP_IO.Charger[i].HV_ON := TRUE;
				MCP_IO.Charger[i].inhibit := FALSE;
				ChargeTime_DB.ChargerDelay_TON[i] (IN := FALSE, PT := ChargeTime_DB.ChargerDelay_PT[i], ET => ChargeTime_DB.ChargerDelay_ET[i]);
				ChargeTime_DB.ChargingTimeElapse_TON[i]  (IN := TRUE, PT := REAL_TO_TIME (1000*MCP_IO.Charger[i].ChargeTime.timeToChargeLoad)); 
			END_IF;
			
			IF ChargeTime_DB.ChargingTimeElapse_TON[i].Q THEN
				StartCharger[i] := FALSE;
				ChargeTime_DB.ChargingTimeElapse_TON[i] (IN := FALSE); 
				//ChargeTime_DB.ChargerDelay_TON[i] (IN := FALSE, PT := ChargeTime_DB.ChargerDelay_PT[i], ET => ChargeTime_DB.ChargerDelay_ET[i]);
			END_IF;
		END_FOR;
		//pfc
		IF ChargeTime_DB.pfcChargerDelay_TON.Q THEN 
			StartCharger[8] := TRUE;
		END_IF;	
		
		IF StartCharger[8] = TRUE THEN 
			GVL.WriteStatetoPLC := E_State.CHARGING;  ///*************** pfc plc will decide the charging time elapse ton.
			ChargeTime_DB.pfcChargerDelay_TON (IN := FALSE, PT := ChargeTime_DB.pfcChargerDelay_PT, ET => ChargeTime_DB.pfcChargerDelay_ET);
			//ChargeTime_DB.ChargingTimeElapse_TON[i]  (IN := TRUE, PT := REAL_TO_TIME (1000*MCP_IO.Charger[i].ChargeTime.timeToChargeLoad)); 
		END_IF
		IF GVL.ReadStateFromPLC = E_State.CHARGECOMPLETE THEN 
			StartCharger[8] := FALSE;
		END_IF
		
		IF ChargingRunOutTMR_TON.Q = TRUE THEN
			Trips_DB.ChargingTimerRunout := TRUE;
			ChargingRunOutTMR_TON (IN := FALSE);
		END_IF;
		
		IF ChargeTime_DB.LongestChargeTime_TON.Q = TRUE THEN 
			ChargeTimeFinished := TRUE;
			StartChargingBroadcast := FALSE;
		
			ChargeTime_DB.LongestChargeTime_TON (IN := FALSE); //reset timer
		END_IF
		
		IF ChargeTimeFinished = TRUE THEN 
			
			FOR i := 1 TO 6 BY 1 DO 
				StartCharger[i] := FALSE;
				ChargeTime_DB.ChargingTimeElapse_TON[i] (IN := FALSE);							
			END_FOR
			
			//pfc
			StartCharger[8] := FALSE; //************************
			
		END_IF
		
		//condition for charge complete
		IF (Permissives_DB.AllChargerEOC = TRUE AND ChargeTimeFinished = TRUE (*all voltage reached*)) OR HMI_DB.ForceToChargCompletePB = TRUE THEN 
			ChargeCompleted := TRUE;
		//ELSE
			//ChargeCompleted := FALSE;
		END_IF
		
//if cap voltage feedback >= charger setpoints && EOC && all timer runout then chargecomplete
		IF ChargeCompleted = TRUE THEN
 
			//MCP_IO.PrefireDiscon.ChargePrefireDisconCap := FALSE; //keep this on, otherwise it will dump

			FOR i := 1 TO 6 BY 1 DO 
				MCP_IO.Charger[i].HV_ON := FALSE; 
				MCP_IO.Charger[i].inhibit := TRUE;
								
				StartCharger[i] := FALSE;
				ChargeTime_DB.ChargingTimeElapse_TON[i] (IN := FALSE);	
			END_FOR;
			ChargeRlyDelayON_Timer ( IN := TRUE, PT := ChargeRlyDelayON_PT);
			StartCharger[8] := FALSE;
		END_IF;
	
		IF ChargeRlyDelayON_Timer.Q = TRUE THEN
			ChargeRlyDelayDONE := TRUE;
		END_IF;
		
		IF ChargeRlyDelayDONE = TRUE THEN
			FOR m := 1 TO 6 BY 1 DO
				//Open all relays
				LCP1_IO.Segment[m].Module[1].CloseChargeRly := FALSE;
				LCP1_IO.Segment[m].Module[2].CloseChargeRly := FALSE;
				LCP1_IO.Segment[m].Module[3].CloseChargeRly := FALSE;
		
				LCP1_IO.Segment[m].Module[1].OpenDumpRly := TRUE;
				LCP1_IO.Segment[m].Module[2].OpenDumpRly := TRUE;
				LCP1_IO.Segment[m].Module[3].OpenDumpRly := TRUE;

			END_FOR;
			ChargeRlyDelayON_Timer ( IN := FALSE, PT := ChargeRlyDelayON_PT);
						
			StartChargingBroadcast := FALSE; // reset the broadcast bit whne all chargers 
			
			eState := E_State.CHARGECOMPLETE;
		END_IF
	
	E_State.CHARGECOMPLETE:
		//close prefire protection disconn
		//MCP_IO.PrefireDiscon.ChargePrefireDisconCap := FALSE;
		//MCP_IO.PrefireDiscon.ClosePrefireDiscon := TRUE;  <- move the when pfc firing and wait 2 sec
		
		//turn on led light
		LCP1_IO.Segment[1].Module[1].ModuleCharged := TRUE;
		ChargeRlyDelayDONE := FALSE;
		ChargeCompleted := FALSE;
		StartChargingBroadcast := FALSE; // reset the broadcast bit whne all chargers 
		ChargedRunOutTMR_TON (IN := TRUE, PT := HMI_DB.RunOutTMR_PT);
		ChargeRlyDelayON_Timer ( IN := FALSE, PT := ChargeRlyDelayON_PT);
		
		GVL.WriteStatetoPLC := E_state.CHARGECOMPLETE; //status to pfc PP
		
		IF HMI_DB.FirePB = TRUE (*AND Permissives_DB.PrefireDisconClosed = TRUE*) THEN 
			//LCP1_IO.Segment[1].Module[1].Fire := TRUE;
			LCP1_IO.Segment[1].Module[1].TriggerScope := TRUE;
			ChargedRunOutTMR_TON (IN := FALSE);
			//and all other shot triggers.
			FirePBpressed := TRUE;
			
			//ELSE
				//LCP1_IO.Segment[1].Module[1].Fire := FALSE;
		END_IF
		
		GVL.Button.FirePBpressed := HMI_DB.FirePB; // send firing signal to pfc
		
		IF FirePBpressed = TRUE THEN 
			//FireToSafeDelayTMR_TON (IN := TRUE, PT := FireToSafeDelayTMR_PT, ET => FireToSafeDelayTMR_ET);
			ShotTrigDelayTMR_TON (IN := TRUE, PT := ShotTrigDelayTMR_PT, ET => ShotTrigDelayTMR_ET);
			ScopeTrigPulseTMR_TON (IN := TRUE, PT := ScopeTrigPulseTMR_PT, ET => ScopeTrigPulseTMR_ET);
			ShotTrigPulseTMR_TON (IN := TRUE, PT := ShotTrigPulseTMR_PT, ET => ShotTrigPulseTMR_ET);
			//LCP1_IO.Segment[1].Module[1].Fire := TRUE;
		END_IF
		
		IF ScopeTrigPulseTMR_TON.Q = TRUE THEN 
			LCP1_IO.Segment[1].Module[1].TriggerScope := FALSE;  //changed to true to keep the pulse on
			//ScopeTrigPulseTMR_TON (IN := FALSE);
		END_IF
		
		IF ShotTrigDelayTMR_TON.Q = TRUE THEN
			LCP1_IO.Segment[1].Module[1].Fire := TRUE;
			ShotFired := TRUE;
			//ShotTrigDelayTMR_TON (IN := FALSE);
		ELSIF ShotTrigPulseTMR_TON.Q = TRUE THEN  // changed to nested elsif
			LCP1_IO.Segment[1].Module[1].Fire := FALSE;
			//LCP1_IO.Segment[1].Module[1].TriggerScope := FALSE;  //need to comment out for scope trigger delay
			//ShotTrigPulseTMR_TON (IN := FALSE);
		END_IF
		
		IF ShotFired = TRUE THEN
			FireToSafeDelayTMR_TON (IN := TRUE, PT := FireToSafeDelayTMR_PT, ET => FireToSafeDelayTMR_ET);
		END_IF
		
		IF FireToSafeDelayTMR_TON.Q = TRUE THEN
			FirePBpressed := FALSE;
			ShotFired := FALSE;
			FireToSafeDelayTMR_TON (IN := FALSE);
			ScopeTrigPulseTMR_TON (IN := FALSE);
			ShotTrigDelayTMR_TON (IN := FALSE);
			ShotTrigPulseTMR_TON (IN := FALSE);
			//LCP1_IO.Segment[1].Module[1].TriggerScope := FALSE;
			eState := E_State.SAFE;
		END_IF;
		
		IF ChargedRunOutTMR_TON.Q = TRUE THEN
			Trips_DB.ChargedTimerRunout := TRUE;
			ChargeTimeFinished := FALSE; //reset chargetime done bit
			ChargedRunOutTMR_TON (IN := FALSE);
			ScopeTrigPulseTMR_TON (IN := FALSE);
			ShotTrigDelayTMR_TON (IN := FALSE);
			ShotTrigPulseTMR_TON (IN := FALSE);
			eState := E_State.ABORT;
		END_IF

	E_State.DUMPING:
	
		MCP_IO.PrefireDiscon.ChargePrefireDisconCap := FALSE;
		MCP_IO.PrefireDiscon.ClosePrefireDiscon := FALSE;
		
		ChargeDelayStart := FALSE;
		FirePBpressed := FALSE;
		ShotTrigDelayTMR_TON (IN := FALSE);
		StartCharWarningTMR_TON (IN := FALSE, PT := StartCharWarningTMR_PT, ET=> StartCharWarningTMR_ET);
		
		ShotTrigDelayTMR_TON (IN := FALSE, PT := ShotTrigDelayTMR_PT, ET => ShotTrigDelayTMR_ET);
		ScopeTrigPulseTMR_TON (IN := FALSE, PT := ScopeTrigPulseTMR_PT, ET => ScopeTrigPulseTMR_ET);
		ShotTrigPulseTMR_TON (IN := FALSE, PT := ShotTrigPulseTMR_PT, ET => ShotTrigPulseTMR_ET);
		
		GVL.WriteStatetoPLC := E_state.DUMPING; //status to pfc PP
		
		// dump all 
		FOR i := 1 TO 6 BY 1 DO 
			MCP_IO.Charger[i].voltageSP := 0.001;
			MCP_IO.Charger[i].inhibit := TRUE;
			MCP_IO.Charger[i].HV_ON := FALSE;
				
			LCP1_IO.Segment[i].Module[1].CloseChargeRly := FALSE;
			LCP1_IO.Segment[i].Module[2].CloseChargeRly := FALSE;
			LCP1_IO.Segment[i].Module[3].CloseChargeRly := FALSE;
		
			LCP1_IO.Segment[i].Module[1].OpenDumpRly := FALSE;
			LCP1_IO.Segment[i].Module[2].OpenDumpRly := FALSE;
			LCP1_IO.Segment[i].Module[3].OpenDumpRly := FALSE;
		END_FOR;
		
		DumpingRunOutTMR_TON (IN := TRUE, PT := DumpingRunOutTMR_PT);
		
		//HMI_DB.CloseChargeRlySW := FALSE;
		//HMI_DB.OpenDumpRlySW := FALSE;
		
		IF DumpingRunOutTMR_TON.Q = TRUE AND Permissives.AllCapsDischarged = TRUE THEN
			eState := E_State.SAFE;
		END_IF

	E_State.ABORT:
				
		//MCP_IO.PrefireDiscon.ChargePrefireDisconCap := FALSE;
		MCP_IO.PrefireDiscon.ClosePrefireDiscon := FALSE;
		
		ChargeDelayStart := FALSE;
		FirePBpressed := FALSE;
		StartCharWarningTMR_TON (IN := FALSE, PT := StartCharWarningTMR_PT, ET=> StartCharWarningTMR_ET);
		
		GVL.WriteStatetoPLC := E_state.ABORT; //status to pfc PP
		
		//dump all
		FOR i := 1 TO 6 BY 1 DO
			MCP_IO.Charger[i].voltageSP := 0.001;
			MCP_IO.Charger[i].inhibit := TRUE;
			MCP_IO.Charger[i].HV_ON := FALSE;
			
		END_FOR
				
		LCP1_IO.Segment[1].Module[1].CloseChargeRly := FALSE;
		LCP1_IO.Segment[1].Module[2].CloseChargeRly := FALSE;
		LCP1_IO.Segment[1].Module[3].CloseChargeRly := FALSE;
		
		LCP1_IO.Segment[1].Module[1].OpenDumpRly := FALSE;
		LCP1_IO.Segment[1].Module[2].OpenDumpRly := FALSE;
		LCP1_IO.Segment[1].Module[3].OpenDumpRly := FALSE;
		
		IF Permissives.SystemIsSafe = TRUE AND Trips_DB.TimerRunOutON = FALSE THEN
			eState := E_State.SAFE;
		END_IF
		
		HMI_DB.CloseChargeRlySW := FALSE;
		HMI_DB.OpenDumpRlySW := FALSE;
		HMI_DB.TurnChrgHVonSW := FALSE;
		HMI_DB.TurnChrgInhibitOffSW := FALSE;
		HMI_DB.TurnOnShotTrigSW := FALSE;
		HMI_DB.TurnOnChargeAlarm := FALSE;
		
		HMI_DB.ClosePrefireDisconSW := FALSE;
		HMI_DB.ChargePrefireDisconCap := FALSE;
		
	E_State.ManualMode:
		GVL.WriteStatetoPLC := E_state.ManualMode; //status to pfc PP
		
		DumpingRunOutTMR_TON (IN := FALSE);
		LCP1_IO.Segment[1].Module[1].CloseChargeRly := HMI_DB.CloseChargeRlySW;
		LCP1_IO.Segment[1].Module[1].OpenDumpRly := HMI_DB.OpenDumpRlySW;
		
		MCP_IO.Charger[1].HV_ON := HMI_DB.TurnChrgHVonSW;
		
		MCP_IO.PrefireDiscon.ClosePrefireDiscon 	:= HMI_DB.ClosePrefireDisconSW;
		MCP_IO.PrefireDiscon.ChargePrefireDisconCap := HMI_DB.ChargePrefireDisconCap;
		
		IF HMI_DB.TurnChrgInhibitOffSW = TRUE THEN 
				MCP_IO.Charger[1].inhibit := FALSE;
			ELSE
				MCP_IO.Charger[1].inhibit := TRUE;
		END_IF
		
		LCP1_IO.Segment[1].Module[1].Fire := HMI_DB.TurnOnShotTrigSW;
		LCP1_IO.Segment[1].Module[1].ModuleCharged := HMI_DB.TurnOnChargeAlarm;
			
		IF HMI_DB.HMI_ManualModeSelected = FALSE THEN
			eState := E_State.SAFE;
		END_IF
	
		//IF HMI_DB.P		MCP_IO.PrefireDiscon.ChargePrefireDisconCap := FALSE;
		//M
		
END_CASE;

IF i > 6 THEN 
	i := 1;
END_IF;	

IF m > 6 THEN 
	m := 1;
END_IF;

END_PROGRAM

// ---- POUs/HMI.TcPOU
PROGRAM HMI
VAR
	eChargerType : E_ChargerType;
	
	//SysCLK					: GETSYSTEMTIME;
	//fileTime				: T_FILETIME;
	LastTimeShot			: STRING;
	ChargeGraphTMR_TON		: TON;
	ChargeGraphTMR_PT		: TIME := ChargeTime_DB.LongestChargeTime_PT + T#10S;
	ChargeGraphTMR_ET		: TIME;
	LongestChargeTIME		: REAL;
	LastTimeShotLog			: BOOL;
	ForceCharCompSatisfied	: BOOL := FALSE;
	
	i : INT := 1;

	LastTimeShotTMR_TON		: TON;
	LastTimeShotTMR_PT		: TIME := T#120H;
	LastTimeShotTMR_ET		: TIME;
	LastTimeShotTMR_REAL	: DWORD;
END_VAR

// if clear all faults, reset abort status
IF HMI_DB.ClearFaultPB = TRUE THEN
	Trips_DB.ChargedTimerRunout := FALSE;
	Trips_DB.ChargingTimerRunout := FALSE;
	Trips_DB.DumpTimerRunout := FALSE;
	Trips_DB.ChargerSummaryFault := FALSE;
	Trips_DB.ShortingSystemUnknown := FALSE;
	VoltMonitor_DB.LossVoltMonitorBoard := FALSE;
END_IF

IF Trips_DB.ChargedTimerRunout = TRUE OR 
	Trips_DB.ChargingTimerRunout = TRUE //OR 
	//Trips_DB.DumpTimerRunout = TRUE 
	THEN
		Trips_DB.TimerRunOutON := TRUE; 
		ELSE
			Trips_DB.TimerRunOutON := FALSE;
		END_IF
FOR i := 1 TO 6 BY 1 DO 
	MCP_IO.Charger[i].ChargerType := Setpoints.TDKLoad[i].eChargerType := HMI_DB.TDKLoad[i].eChargerType;
	IF MCP_IO.Charger[i].ChargerType = E_ChargerType.TDK12kV THEN 
		HMI_DB.TDKLoad[i].PSratedV := 12;
		ELSIF MCP_IO.Charger[i].ChargerType = E_ChargerType.TDK30kV THEN
			HMI_DB.TDKLoad[i].PSratedV := 30;
		ELSIF MCP_IO.Charger[i].ChargerType = E_ChargerType.TDK50kV THEN
			HMI_DB.TDKLoad[i].PSratedV := 50;
	END_IF
END_FOR;

LastTimeShotTMR_TON (IN := TRUE, PT := LastTimeShotTMR_PT, ET => LastTimeShotTMR_ET);

IF (Sequence.eState = E_State.CHARGECOMPLETE) AND HMI_DB.FirePB = TRUE THEN 
	//SysCLK (timeLoDW => fileTime.dwLowDateTime, timeHiDW => fileTime.dwHighDateTime);
	//LastTimeShot := SYSTEMTIME_TO_STRING( FILETIME_TO_SYSTEMTIME( fileTime ) );	
	LastTimeShotTMR_TON (IN := FALSE, PT := LastTimeShotTMR_PT, ET => LastTimeShotTMR_ET);
	HMI_DB.LastTimeShotLog := TRUE;	
	ELSE
		HMI_DB.LastTimeShotLog := FALSE;
END_IF

LastTimeShotTMR_REAL := TIME_TO_DWORD (LastTimeShotTMR_ET)/1000;

IF (Sequence.eState = E_State.CHARGECOMPLETE OR Sequence.eState = E_State.CHARGING) THEN
	ChargeGraphTMR_TON (IN:= TRUE, PT:= ChargeGraphTMR_PT, ET => ChargeGraphTMR_ET);
	ELSE
		ChargeGraphTMR_TON (IN:= FALSE);
END_IF

LongestChargeTIME := TIME_TO_REAL (ChargeTime_DB.LongestChargeTime_ET)/1000;

//forced shoot threshold condition
//***************note: we are only using charger 1****** 
IF (MCP_IO.Charger[1].voltageFeedback >= 0.8*Setpoints.TDKLoad[1].RequiredChargedV*1000) OR 
	(LCP1_IO.Segment[1].Module[1].VoltageFeedback >= 0.8*Setpoints.TDKLoad[1].RequiredChargedV*1000) 
	THEN  //might need to do ABS for -2
		ForceCharCompSatisfied := TRUE;
ELSE
	ForceCharCompSatisfied := FALSE;
END_IF

(********************HMI logic for csv logging status***************)
IF P_TextModeWrite.bBusy = TRUE THEN 
	HMI_DB.CSV_loggingBusy := TRUE;
	ELSE
		HMI_DB.CSV_loggingBusy := FALSE;
END_IF

IF P_TextModeWrite.bError = TRUE THEN 
	HMI_DB.CSV_loggingError := TRUE;
	ELSE
		HMI_DB.CSV_loggingError := FALSE;
END_IF

//IF P_TextModeWrite.step = 10 AND P_TextModeWrite.bBusy = FALSE THEN 
	//HMI_DB.CSV_loggingDone := TRUE;
	//ELSIF P_TextModeWrite.step = 0 AND P_TextModeWrite.bBusy = TRUE THEN
		//HMI_DB.CSV_loggingDone := FALSE;
//END_IF

//Status light for saving csv buffer
IF P_TextModeWrite.SaveBuff = TRUE THEN 
	HMI_DB.FillingBuffer := TRUE;
	ELSE
		HMI_DB.FillingBuffer := FALSE;
END_IF

IF P_TextModeWrite.SaveCSV = FALSE AND P_TextModeWrite.step = 10 THEN 
	HMI_DB.CSV_loggingDone := TRUE;
	ELSIF (P_TextModeWrite.SaveCSV = TRUE OR P_TextModeWrite.SaveBuff = TRUE)  THEN
		HMI_DB.CSV_loggingDone := FALSE;
END_IF

HMI_DB.FireDelayTMR_PT := REAL_TO_TIME (HMI_DB.FireDelayTMR_REAL *1000);  // delay firing between pfc firing and shot disconnect

IF i > 6 THEN 
	i := 1;
END_IF

END_PROGRAM

// ---- POUs/csv/P_TextModeWrite.TcPOU
(* Writing of CSV file in text mode. None of the field value is containing any non-printing control characters like line feed, carriage return, quotation marks, semicolon... *)
PROGRAM P_TextModeWrite
VAR_INPUT
	bWrite			: BOOL := FALSE;(* Rising edge starts program execution *)
END_VAR
VAR
	//bWrite			: BOOL := FALSE;(* Rising edge starts program execution *)
	timer_TON		: TON;
	timer_PT		: TIME;
	timer_ET		: TIME;
	timestamp		: REAL;
	SysCLK			: GETSYSTEMTIME;
	fileTime		: T_FILETIME;
	location		: T_MaxString := 'C:\CSVdata\';
	fileType		: T_MaxString := '.csv';
	filename		: STRING;
	filename_full	: T_MaxString;
	filename_short	: T_MaxString;
	sNetId			: T_AmsNetId := '';	(* TwinCAT system network address *)
	sFileName		: T_MaxString := 'C:\CSVdata\ChargerVClog.csv';(* CSV destination file path and name *)
	sCSVLine		: T_MaxString := '';(* Single CSV text line (row, record), we are using string as record buffer (your are able to see created fields) *)
	sCSVField		: T_MaxString := '';(* Single CSV field value (column, record field) *)
	bBusy			: BOOL;
	bError			: BOOL;
	nErrId			: UDINT;
	nRow	 		: UDINT 	:= 0;(* Row number (record) *)
	nColumn			: UDINT 	:= 0;(* Column number (record field) *)
	hFile			: UINT		:= 0;(* File handle of the source file *)
	step			: DWORD 	:= 0;
	fbFileOpen		: FB_FileOpen;(* Opens file *)
	fbFileClose		: FB_FileClose;(* Closes file *)
	fbFilePuts		: FB_FilePuts;(* Writes one record (line) *)
	fbWriter		: FB_CSVMemBufferWriter;(* Helper function block used to create CSV data bytes (single record line) *)
	
	//eState 					: E_State;
	csvW_RebounceTMR_TON	: TON;
	csvW_RebounceTMR_PT		: TIME := T#500MS;
	StartLogging_ONS		: BOOL;
	i 						: UDINT := 0;
	SamplingTMR_TON 		: TON;
	SamplingTMR_PT			: TIME := T#1S;
	SamplingTMR_ET			: TIME;
	SaveCSV					: BOOL := FALSE;
	SaveBuff			: BOOL := FALSE;
	
	database		: ARRAY[0..GVL.MAX_CSV_ROWS, 0..GVL.MAX_CSV_COLUMNS ] OF STRING(GVL.MAX_CSV_FIELD_LENGTH) :=[ (* Source PLC database *)
	'0_0', '0_1', '0_2', '0_3', '0_4', '0_5',
	'1_0', '1_1', '1_2', '1_3', '1_4', '1_5',
	'2_0', '2_1', '2_2', '2_3', '2_4', '2_5',
	'3_0', '3_1', '3_2', '3_3', '3_4', '3_5',
	'4_0', '4_1', '4_2', '4_3', '4_4', '4_5',
	'5_0', '5_1', '5_2', '5_3', '5_4', '5_5'];
	


END_VAR



SysCLK (timeLoDW => fileTime.dwLowDateTime, timeHiDW => fileTime.dwHighDateTime);

filename_full := DT_TO_STRING (FILETIME_TO_DT (fileTIME));

//filename_short := DELETE (DELETE (RIGHT (filename_full, 19), 1, 14), 1, 16);// LEFT (STR := filename, 35);
//sFileName := CONCAT (STR1 := 'C:\CSVdata\', STR2 := filename);
//filename := CONCAT (STR1 := filename_short, STR2 := fileType); //incrementing file name
//sFileName := CONCAT (STR1 := location, STR2 := filename);
CASE step OF
	0:	(* Wait for rising edge at bWrite variable *)
		IF bWrite THEN
			bWrite 	:= FALSE;
			bBusy 	:= TRUE;
			bError	:= FALSE;
			nErrId	:= 0;
			hFile	:= 0;
			nRow	:= 0;
			nColumn	:= 0;
			step 	:= 1;
		END_IF

	1:	(* Open source file *)
		fbFileOpen(  bExecute := FALSE  );
		
		filename_short := DELETE (DELETE (RIGHT (filename_full, 19), 1, 14), 1, 16);// LEFT (STR := filename, 35);
		filename := CONCAT (STR1 := filename_short, STR2 := fileType); //incrementing file name
		sFileName := CONCAT (STR1 := location, STR2 := filename);
		
		fbFileOpen( sNetId := sNetId, sPathName := sFileName, nMode := FOPEN_MODEWRITE OR FOPEN_MODETEXT,(* Open file in TEXT mode! *)
					ePath := PATH_GENERIC, bExecute := TRUE );
		step := 2;

	2:(* Wait until open not busy *)
		fbFileOpen( bExecute := FALSE, bError => bError, nErrID => nErrID, hFile => hFile );
		IF NOT fbFileOpen.bBusy THEN
			IF NOT fbFileOpen.bError THEN
				step := 3;
			ELSE(* Error: file not found? *)
				step := 100;
			END_IF
		END_IF

	3:(* Convert one PLC record to CSV format *)
		sCSVLine := '';
		fbWriter.eCmd := eEnumCmd_First;(* Write first field value *)
		IF nRow <= GVL.MAX_CSV_ROWS THEN
		
			FOR nColumn := 0 TO GVL.MAX_CSV_COLUMNS BY 1 DO

				sCSVField := STRING_TO_CSVFIELD( database[ nRow, nColumn ], FALSE );(* TODO: Get field value from your application *)

				(* Add new field to the record buffer *)
				fbWriter( 	pBuffer := ADR( sCSVLine ), cbBuffer := SIZEOF( sCSVLine ) - 1, putValue := sCSVField, pValue := 0, cbValue := 0,
							bCRLF := ( nColumn = GVL.MAX_CSV_COLUMNS ) );(* bCRLF == TRUE => Write CRLF after the last field value *)
				IF fbWriter.bOk THEN
					fbWriter.eCmd := eEnumCmd_Next;(* Write next field value *)
				ELSE(* Error *)
					step := 100;
					RETURN;
				END_IF

			END_FOR(* FOR nColumn := 0... *)

			(* FB_FilePuts adds allready CR (carriage return) to the written line.
			We have to replace the $R$L characters with $L character to avoid double CR. *)
			IF RIGHT( sCSVLine, 2 ) = '$R$L' THEN
				sCSVLine := REPLACE( sCSVLine, '$L', 2, LEN( sCSVLine ) - 1 );
			END_IF

			nRow := nRow + 1;(* Increment number of created records (rows) *)

			step := 4;(* Write record to the file *)

		ELSE(* All rows written => Close file *)
			step := 10;
		END_IF

	4:	(* Write single text line *)
		fbFilePuts( bExecute := FALSE );
		fbFilePuts( sNetId := sNetId, hFile := hFile, sLine := sCSVLine, bExecute := TRUE );
		step := 5;

	5:(* Wait until write not busy *)
		fbFilePuts( bExecute := FALSE, bError => bError, nErrID => nErrID );
		IF NOT fbFilePuts.bBusy THEN
			IF NOT fbFilePuts.bError THEN
				step := 3;(* Write next record *)
			ELSE(* Error *)
				step := 100;
			END_IF
		END_IF

	10:	(* Close source file *)
		fbFileClose( bExecute := FALSE );
		fbFileClose( sNetId := sNetId, hFile := hFile, bExecute := TRUE );
		step := 11;

	11:(* Wait until close not busy *)
		fbFileClose( bExecute := FALSE, bError => bError, nErrID => nErrID );
		IF ( NOT fbFileClose.bBusy ) THEN
			hFile := 0;
			step := 100;
		END_IF

	100: (* Error or ready step => cleanup *)
		IF ( hFile <> 0 ) THEN
			step := 10; (* Close the source file *)
		ELSE
			bBusy := FALSE;
			step := 0;	(* Ready *)
		END_IF

END_CASE



//logging logic
//start storing buffer when charge pb is pressed. 
//when charge done, convert data into csv.
IF (*Sequence.eState = E_State.CHARGING*) HMI_DB.ChargePB = TRUE THEN 
	//StartLogging_ONS := TRUE;
	SaveBuff := TRUE; 
	//ELSIF Sequence.eState = E_State.SAFE THEN
		//bWrite := FALSE;
		//step := 10;
		//fbFileClose( bExecute := FALSE );
		//fbFileClose( sNetId := sNetId, hFile := hFile, bExecute := TRUE );
END_IF


//logging data - either need a timer to store the database buffer or user a timer to call the function.
IF SaveBuff = TRUE THEN 
	timer_TON (IN:= TRUE, PT := (ChargeTime_DB.LongestChargeTime_PT + HMI_DB.RunOutTMR_PT + T#10S), ET => timer_ET);
	IF SamplingTMR_TON.Q = FALSE THEN
		SamplingTMR_TON (IN := TRUE, PT := SamplingTMR_PT, ET => SamplingTMR_ET);
		//csvW_RebounceTMR_TON(IN := TRUE, PT := csvW_RebounceTMR_PT );
		ELSE 
			SamplingTMR_TON (IN := FALSE, PT := SamplingTMR_PT);
	END_IF 
ELSE
		SamplingTMR_TON (IN := FALSE, PT := SamplingTMR_PT);
		timer_TON (IN:= FALSE);
END_IF

timestamp := TIME_TO_REAL (timer_ET)/1000; 
	
IF (i <= GVL.MAX_CSV_ROWS) AND SamplingTMR_TON.Q = TRUE THEN 
	database[i, 0] := REAL_TO_STRING(timestamp);
	database[i, 1] := REAL_TO_STRING(MCP_IO.Charger[1].voltageFeedback);
	database[i, 2] := REAL_TO_STRING(MCP_IO.Charger[1].currentFeedback);
		
	//uncomment for testing purposes
		//Input.R1_08_00 := Input.R1_08_00 + 10 ;
		//Input.R1_08_01 := Input.R1_08_00 + 100 ;
		i := i + 1;
		SamplingTMR_TON.IN := FALSE;

ELSIF (i > GVL.MAX_CSV_ROWS) OR ((Sequence.eState = E_State.ABORT OR HMI_DB.FirePB = TRUE OR HMI_DB.DumpPB = TRUE OR HMI_DB.AbortPB = TRUE) AND i <> 0) THEN 
	SaveCSV := TRUE;
	SaveBuff := FALSE; 
	SamplingTMR_TON.IN := FALSE;
	i := 0;
	ELSE
		SamplingTMR_TON.IN := FALSE;
END_IF

IF SaveCSV = TRUE THEN 
	bWrite := TRUE;
	csvW_RebounceTMR_TON(IN := TRUE, PT:= csvW_RebounceTMR_PT);
END_IF

IF csvW_RebounceTMR_TON.Q = TRUE THEN 
	SaveCSV := FALSE;
	bWrite := FALSE;
	csvW_RebounceTMR_TON(IN := FALSE, PT:= csvW_RebounceTMR_PT);
END_IF

	//bWrite := FALSE;
	//step := 10;
	//fbFileClose( bExecute := FALSE );
	//fbFileClose( sNetId := sNetId, hFile := hFile, bExecute := TRUE );

END_PROGRAM

// ---- POUs/Heartbeat.TcPOU
PROGRAM Heartbeat
VAR
	start_TON				: TON;
	start_TON_et 			: TIME;
	reset_TON 				: TON;
	reset_TON_et 			: TIME;
	screen_refresh_pulse 	: BOOL;
	
	pulse_1Hz_Start_TON		: TON;
	pulse_1Hz_Start_PT		: TIME := T#125MS;
	pulse_1Hz_Reset_TON		: TON;
	pulse_1Hz_Reset_PT		: TIME := T#125MS;
	pulse_1Hz				: BOOL;
END_VAR

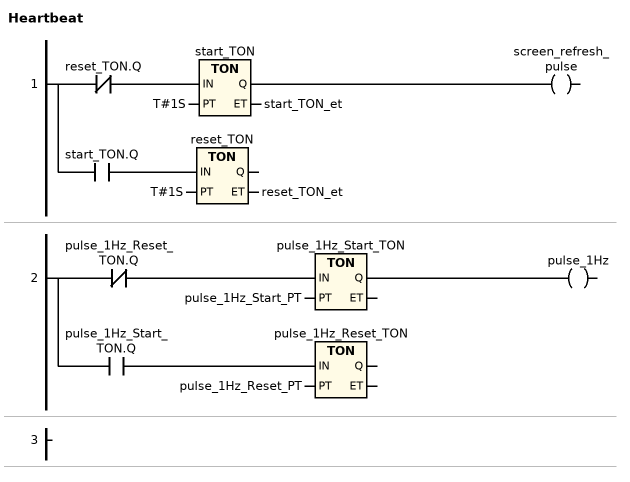
// NETWORK 1
start_TON(IN := NOT reset_TON.Q, PT := T#1S, ET => start_TON_et); // TON
screen_refresh_pulse := start_TON.Q;
reset_TON(IN := start_TON.Q, PT := T#1S, ET => reset_TON_et); // TON

// NETWORK 2
pulse_1Hz_Start_TON(IN := NOT pulse_1Hz_Reset_TON.Q, PT := pulse_1Hz_Start_PT); // TON
pulse_1Hz := pulse_1Hz_Start_TON.Q;
pulse_1Hz_Reset_TON(IN := pulse_1Hz_Start_TON.Q, PT := pulse_1Hz_Reset_PT); // TON

// NETWORK 3

END_PROGRAM

// ---- POUs/Alarms.TcPOU
PROGRAM Alarms
VAR
	bWarning : BOOL;
	bConfirm : BOOL;
	alarms : ARRAY[0..32] OF Alarms_FB;
	
END_VAR

// Alarm Word 1 - MCP Alarms
//MCP Alarms

Alarms_DB.MCP.AlarmWord.0 := Trips_DB.EStopPBpressed;
Alarms_DB.MCP.AlarmWord.1 := Trips_DB.CageDoorNotClose;
Alarms_DB.MCP.AlarmWord.2 := Trips_DB.ShortingSystemUnknown;
Alarms_DB.MCP.AlarmWord.3 := Permissives_DB.PrefireDisconClosed;
Alarms_DB.MCP.AlarmWord.4 := MCP_IO.Charger[1].SummaryFaulted;
Alarms_DB.MCP.AlarmWord.5 := Permissives_DB.PrefireDisconOpen;
//Alarms_DB.MCP.AlarmWord.6 := MCP_IO.Charger[3].SummaryFaulted;
//Alarms_DB.MCP.AlarmWord.7 := MCP_IO.Charger[4].SummaryFaulted;
//Alarms_DB.MCP.AlarmWord.8 := MCP_IO.Charger[5].SummaryFaulted;
//Alarms_DB.MCP.AlarmWord.9 := MCP_IO.Charger[6].SummaryFaulted;
Alarms_DB.MCP.AlarmWord.10 := HMI_DB.ForceToChargCompletePB;
Alarms_DB.MCP.AlarmWord.11 := VoltMonitor_DB.LossVoltMonitorBoard;
Alarms_DB.MCP.AlarmWord.12 := Trips_DB.ChargedTimerRunout;
Alarms_DB.MCP.AlarmWord.13 := Trips_DB.ChargingTimerRunout;
Alarms_DB.MCP.AlarmWord.14 := HMI_DB.LastTimeShotLog;
Alarms_DB.MCP.AlarmWord.15 := HMI.ForceCharCompSatisfied;

//Alarm Word 1 msg
//IE: alarms[299](evtEntry:= Tc_Events.AlarmWord11.b4, bEvt:= gvl.test, bConfirm:= bConfirm);
alarms[0](evtEntry:= Tc_Events.AlarmWord1.b0, bEvt:= Alarms_DB.MCP.AlarmWord.0, bConfirm:= bConfirm);
alarms[1](evtEntry:= Tc_Events.AlarmWord1.b1, bEvt:= Alarms_DB.MCP.AlarmWord.1, bConfirm:= bConfirm);
alarms[2](evtEntry:= Tc_Events.AlarmWord1.b2, bEvt:= Alarms_DB.MCP.AlarmWord.2, bConfirm:= bConfirm);
alarms[3](evtEntry:= Tc_Events.AlarmWord1.b3, bEvt:= Alarms_DB.MCP.AlarmWord.3, bConfirm:= bConfirm);
alarms[4](evtEntry:= Tc_Events.AlarmWord1.b4, bEvt:= Alarms_DB.MCP.AlarmWord.4, bConfirm:= bConfirm);
alarms[5](evtEntry:= Tc_Events.AlarmWord1.b5, bEvt:= Alarms_DB.MCP.AlarmWord.5, bConfirm:= bConfirm);
alarms[6](evtEntry:= Tc_Events.AlarmWord1.b6, bEvt:= Alarms_DB.MCP.AlarmWord.6, bConfirm:= bConfirm);
alarms[7](evtEntry:= Tc_Events.AlarmWord1.b7, bEvt:= Alarms_DB.MCP.AlarmWord.7, bConfirm:= bConfirm);
alarms[8](evtEntry:= Tc_Events.AlarmWord1.b8, bEvt:= Alarms_DB.MCP.AlarmWord.8, bConfirm:= bConfirm);
alarms[9](evtEntry:= Tc_Events.AlarmWord1.b9, bEvt:= Alarms_DB.MCP.AlarmWord.9, bConfirm:= bConfirm);
alarms[0](evtEntry:= Tc_Events.AlarmWord1.b10, bEvt:= Alarms_DB.MCP.AlarmWord.10, bConfirm:= bConfirm);
alarms[11](evtEntry:= Tc_Events.AlarmWord1.b11, bEvt:= Alarms_DB.MCP.AlarmWord.11, bConfirm:= bConfirm);
alarms[12](evtEntry:= Tc_Events.AlarmWord1.b12, bEvt:= Alarms_DB.MCP.AlarmWord.12, bConfirm:= bConfirm);
alarms[13](evtEntry:= Tc_Events.AlarmWord1.b13, bEvt:= Alarms_DB.MCP.AlarmWord.13, bConfirm:= bConfirm);
alarms[14](evtEntry:= Tc_Events.AlarmWord1.b14, bEvt:= Alarms_DB.MCP.AlarmWord.14, bConfirm:= bConfirm);
alarms[15](evtEntry:= Tc_Events.AlarmWord1.b15, bEvt:= Alarms_DB.MCP.AlarmWord.15, bConfirm:= bConfirm);

// Alarm Word 2 - Section 1 Alarms
(*Alarms_DB.Section1.AlarmWord.0 := Trips_DB.Section[1].SystemTripped;
Alarms_DB.Section1.AlarmWord.1 := Trips_DB.Section[1].LossPneumaticPressure;
Alarms_DB.Section1.AlarmWord.2 := Trips_DB.Section[1].Peak.ChargeRelay1_Failed;
Alarms_DB.Section1.AlarmWord.3 := Trips_DB.Section[1].Peak.ChargeRelay2_Failed;
Alarms_DB.Section1.AlarmWord.4 := Trips_DB.Section[1].Peak.DumpRelay1_Failed;
Alarms_DB.Section1.AlarmWord.5 := Trips_DB.Section[1].Peak.DumpRelay2_Failed;
Alarms_DB.Section1.AlarmWord.6 := Trips_DB.Section[1].Sust.ChargeRelay1_Failed;
Alarms_DB.Section1.AlarmWord.7 := Trips_DB.Section[1].Sust.ChargeRelay2_Failed;
Alarms_DB.Section1.AlarmWord.8 := Trips_DB.Section[1].Sust.DumpRelay1_Failed;
Alarms_DB.Section1.AlarmWord.9 := Trips_DB.Section[1].Sust.DumpRelay2_Failed;
Alarms_DB.Section1.AlarmWord.10 := Trips_DB.Section[1].LossDCPower;


// Alarm Word 2 - Msg
alarms[16](evtEntry:= Tc_Events.AlarmWord2.b0, bEvt:= Alarms_DB.Section1.AlarmWord.0, bConfirm:= bConfirm);
alarms[17](evtEntry:= Tc_Events.AlarmWord2.b1, bEvt:= Alarms_DB.Section1.AlarmWord.1, bConfirm:= bConfirm);
alarms[18](evtEntry:= Tc_Events.AlarmWord2.b2, bEvt:= Alarms_DB.Section1.AlarmWord.2, bConfirm:= bConfirm);
alarms[19](evtEntry:= Tc_Events.AlarmWord2.b3, bEvt:= Alarms_DB.Section1.AlarmWord.3, bConfirm:= bConfirm);
alarms[20](evtEntry:= Tc_Events.AlarmWord2.b4, bEvt:= Alarms_DB.Section1.AlarmWord.4, bConfirm:= bConfirm);
alarms[21](evtEntry:= Tc_Events.AlarmWord2.b5, bEvt:= Alarms_DB.Section1.AlarmWord.5, bConfirm:= bConfirm);
alarms[22](evtEntry:= Tc_Events.AlarmWord2.b6, bEvt:= Alarms_DB.Section1.AlarmWord.6, bConfirm:= bConfirm);
alarms[23](evtEntry:= Tc_Events.AlarmWord2.b7, bEvt:= Alarms_DB.Section1.AlarmWord.7, bConfirm:= bConfirm);
alarms[24](evtEntry:= Tc_Events.AlarmWord2.b8, bEvt:= Alarms_DB.Section1.AlarmWord.8, bConfirm:= bConfirm);
alarms[25](evtEntry:= Tc_Events.AlarmWord2.b9, bEvt:= Alarms_DB.Section1.AlarmWord.9, bConfirm:= bConfirm);
alarms[26](evtEntry:= Tc_Events.AlarmWord2.b10, bEvt:= Alarms_DB.Section1.AlarmWord.10, bConfirm:= bConfirm);
//alarms[27] - spare
//alarms[28] - spare
//alarms[29] - spare
//alarms[30] - spare
//alarms[31] - spare
*)

//Clear Alarm Word
IF bConfirm THEN
	Alarms_DB.MCP.AlarmWord := 0;
	Alarms_DB.Segment1.AlarmWord := 0;
	
	(*Alarms_DB.Coil3.AlarmWord := 0;
	Alarms_DB.Coil4.AlarmWord := 0;
	Alarms_DB.Coil5.AlarmWord := 0;
	Alarms_DB.Coil6.AlarmWord := 0;
	Alarms_DB.Coil7.AlarmWord := 0;
	Alarms_DB.Coil8.AlarmWord := 0;
	Alarms_DB.Coil9.AlarmWord := 0;
	Alarms_DB.Coil10.AlarmWord := 0;
	Alarms_DB.AlarmWord_11.AlarmWord := 0;
	Alarms_DB.AlarmWord_22.AlarmWord := 0;
	Alarms_DB.AlarmWord_23.AlarmWord := 0;
	Alarms_DB.AlarmWord_24.AlarmWord := 0;
	Alarms_DB.AlarmWord_25.AlarmWord := 0;
	Alarms_DB.AlarmWord_26.AlarmWord := 0;
	Alarms_DB.AlarmWord_27.AlarmWord := 0;
	*)
END_IF;

END_PROGRAM

// ---- POUs/AnalogConversion_obs.TcPOU
PROGRAM AnalogConversion_obs
VAR
	i					: INT := 1; //charger 1-6
	j					: INT := 1;  // section 1 - 4 
	k					: INT := 1;  // cap 1-10
	m					: INT := 1; //form cap 1-12
END_VAR

//MCP Charger 
//Analog Input
FOR i := 1 TO 6 BY 1 DO 
	//MCP_IO.Charger[i].voltageSP := (HMI_DB.TDKLoad[i].RequiredChargedV *1000);
	MCP_IO.Charger[i].voltageSP := (1000*Setpoints.TDKLoad[i].RequiredChargedV);
END_FOR

//charger 1 is 30kV *************************************************************************************
MCP_IO.Charger[1].voltageFeedback_norm := Norm_x (raw_input := INT_TO_REAL (MCP_IO.Charger[1].voltageFeedback_raw),
														x_max := 32767,
														x_min := 0);
MCP_IO.Charger[1].voltageFeedback := (30000 - 0) * ADC_10V(normal_input := MCP_IO.Charger[1].voltageFeedback_norm,
															x_max := 10,
															x_min := 0);
															
	MCP_IO.Charger[1].currentFeedback_norm := Norm_x (raw_input := INT_TO_REAL (MCP_IO.Charger[1].currentFeedback_raw),
														x_max := 32767,
														x_min := 0);
	// 30kV charger max current output is 0.6A													
	MCP_IO.Charger[1].currentFeedback := (0.6 - 0) * ADC_10V(normal_input := MCP_IO.Charger[1].currentFeedback_norm,
															x_max := 10,
															x_min := 0);																							
//*************************************************************************************

FOR i := 2 TO 6 BY 1 DO
	
	MCP_IO.Charger[i].ChargerType_12kV := NOT MCP_IO.Charger[i].ChargerType_50kV;
	//voltage
	MCP_IO.Charger[i].voltageFeedback_norm := Norm_x (raw_input := INT_TO_REAL (MCP_IO.Charger[i].voltageFeedback_raw),
														x_max := 32767,
														x_min := 0);
	//current																									
	MCP_IO.Charger[i].currentFeedback_norm := Norm_x (raw_input := INT_TO_REAL (MCP_IO.Charger[i].currentFeedback_raw),
														x_max := 32767,
														x_min := 0);
	//50kV chargers feedback
	//if 50kV config selected
	IF MCP_IO.Charger[i].ChargerType_50kV = TRUE THEN 
		//50kv
		MCP_IO.Charger[i].voltageFeedback := (EngVal.Max_50kVChargerVoltage - EngVal.Min_50kVChargerVoltage) * ADC_10V(
																							normal_input := MCP_IO.Charger[i].voltageFeedback_norm,
																							x_max := 10,
																							x_min := 0);

		MCP_IO.Charger[i].currentFeedback := (EngVal.Max_50kVChargerCurrent - EngVal.Min_50kVChargerCurrent) * ADC_10V(
																							normal_input := MCP_IO.Charger[i].currentFeedback_norm,
																							x_max := 10,
																							x_min := 0);
		//12kv
	ELSIF MCP_IO.Charger[i].ChargerType_12kV = TRUE THEN
		MCP_IO.Charger[i].voltageFeedback := (EngVal.Max_12kVChargerVoltage - EngVal.Min_12kVChargerVoltage) * ADC_10V(normal_input := MCP_IO.Charger[i].voltageFeedback_norm,
																														x_max := 10,
																														x_min := 0);
		MCP_IO.Charger[i].currentFeedback := (EngVal.Max_12kVChargerCurrent - EngVal.Min_12kVChargerCurrent) * ADC_10V(
																							normal_input := MCP_IO.Charger[i].currentFeedback_norm,
																							x_max := 10,
																							x_min := 0);										
	END_IF;	
END_FOR;

//Analog Output
//voltageSP = Required Charge Voltage**
//limit for charing the cap

//Charger 1 is 30kV *************************************
IF MCP_IO.Charger[1].voltageSP >= (12000) THEN
			MCP_IO.Charger[1].voltageSP := 10000; //limit at 35kV
		ELSIF MCP_IO.Charger[1].voltageSP <= 0 THEN
			MCP_IO.Charger[1].voltageSP := 0; //limit at 0V
		END_IF; 

//prepare output signal for 30kV chargers.  //**Setpoints.RequiredChargedV -> MCP_IO.Charger.voltageSP **
MCP_IO.Charger[1].voltageSP_norm := Norm_x (raw_input := (MCP_IO.Charger[1].voltageSP), 
												x_max := 30000,
												x_min := 0);
		
MCP_IO.Charger[1].voltageSP_raw := AQ (norm_input := MCP_IO.Charger[1].voltageSP_norm, 
												x_max := 10,
												x_min := 0); 
	
												
//limite for output sigal (<= 10V)  this should not happen
IF MCP_IO.Charger[1].voltageSP_raw >= 32767 THEN 
	MCP_IO.Charger[1].voltageSP_raw := 32767; 										
END_IF;
//*******************************************************

//FOR i := 1 TO 8 BY 1 DO
FOR i := 2 TO 6 BY 1 DO	
	
	//if 50kV config selected
	IF MCP_IO.Charger[i].ChargerType_50kV = TRUE THEN 
		//set limits of charger voltage input 
		IF MCP_IO.Charger[i].voltageSP >= (EngVal.UpperLimit50kVCaps) THEN
			MCP_IO.Charger[i].voltageSP := 35000; //limit at 35kV
		ELSIF MCP_IO.Charger[i].voltageSP <= 0 THEN
			MCP_IO.Charger[i].voltageSP := 0; //limit at 0V
		END_IF; 
		
		(*//set limites of charger voltage input from HMI input
		IF 1000*(Setpoints.TDKLoad[i].RequiredChargedV) >= EngVal.UpperLimit50kVCaps THEN
			Setpoints.TDKLoad[i].RequiredChargedV := (EngVal.UpperLimit50kVCaps/1000); //limit at 35kv
		ELSIF Setpoints.TDKLoad[i].RequiredChargedV <= 0 THEN
			Setpoints.TDKLoad[i].RequiredChargedV :=0 ;
		END_IF*)
		
	//prepare output signal for 50kV chargers.
		MCP_IO.Charger[i].voltageSP_norm := Norm_x (raw_input :=(MCP_IO.Charger[i].voltageSP), 
												x_max := EngVal.Max_50kVChargerVoltage,
												x_min := EngVal.Min_50kVChargerVoltage);	
												
		MCP_IO.Charger[i].voltageSP_raw := AQ (norm_input := MCP_IO.Charger[i].voltageSP_norm, 
												x_max := 10,
												x_min := 0);
	END_IF;
		
	//if 12kV config selected
	IF MCP_IO.Charger[i].ChargerType_12kV = TRUE THEN
		//set limits of charger voltage input 
		IF MCP_IO.Charger[i].voltageSP <= 0 THEN
			MCP_IO.Charger[i].voltageSP := ABS(MCP_IO.Charger[i].voltageSP);
		END_IF
		
		IF MCP_IO.Charger[i].voltageSP >= (EngVal.UpperLimit12kVCaps) THEN
			MCP_IO.Charger[i].voltageSP := 10000; //limit at 10kV
		END_IF;
		
